bStoppingWeight3 := (iWeightCase = 20 AND P05_Weight.fbWeightStation.bWeighingCycleDone AND NOT P05_Weight.fbWeightStation.bCanReleaseForms);
bStoppingWeight4 := tonbCapSorterOrCapSorterDragError.Q; //Opóźnienie zeby wagi dkończyły cykl
//bStoppingWeight4 := stCapSorterRead.eError.bError OR P08_CapSorter.fbCapSorterDragStation.eState = E_Station.eError;

tonStoppingBottleTransfer1	(IN:=iBottleTransferCase = 2, PT:=T#3S);


IF stCapSorterRead.eError.bError THEN
	bCapSorterError := TRUE;
END_IF
tonbCapSorterError(IN:=bCapSorterError,	PT:=T#5S);


CASE iStoppingCase OF
	
	0: //init
		iStoppingCase										:= 10;
		
	10:
		IF
		//P01_BottleFeeder.fbBottleFeeder.eState<=10 AND					
		//P01_BottleFeeder.fbTurnTable.eState<=10 AND	
		//P01_BottleFeeder.fbGateBottleFeeder.eState<=13 AND
		//P01_PucksInserter.fbPucksInserter.eState<=10 AND					
		////P01_PucksInserter.fbTurnTable.eState<=10 AND	
		//P01_PucksInserter.fbGatePucksInserter.eState<=13 AND				
 		//(
		//stBottleSorterRead.ePackMLAutoState <> Tc3_PackML.E_PMLState.ePMLState_STOPPED OR
		//stBottleSorterRead.ePackMLAutoState <> Tc3_PackML.E_PMLState.ePMLState_IDLE OR
		//stBottleSorterRead.ePackMLAutoState <> Tc3_PackML.E_PMLState.ePMLState_RESETTING OR
		//stBottleSorterRead.ePackMLAutoState <> Tc3_PackML.E_PMLState.ePMLState_ABORTED OR
		//stBottleSorterRead.ePackMLAutoState <> Tc3_PackML.E_PMLState.ePMLState_ABORTING OR
		//NOT stBottleSorterRead.bEnable OR bBottleSorterDisable
		//) AND
		P01_Gates.fbGateBeforeDispencers.eState<=13 AND					
		P01_Gates.fbGateRobot.eState<=13 AND					
		P02_Dispencers.fbDispencersDragRightStation.eState<=10 AND
		P02_Dispencers.fbDispencersDragLeftStation.eState<=10 AND	
		P02_Dispencers.fbDispencer1.eState <= 10 AND
		P02_Dispencers.fbDispencer2.eState <= 10 AND
		P02_Dispencers.fbDispencer3.eState <= 10 AND
		P02_Dispencers.fbDispencer4.eState <= 10 AND
		P02_Dispencers.fbDispencersCatch1Station.eState <= 10 AND
		P02_Dispencers.fbDispencersCatch2Station.eState <= 10 AND
		P02_Dispencers.fbDispencersCatch3Station.eState <= 10 AND
		P02_Dispencers.fbDispencersCatch4Station.eState <= 10 AND	
		( //Namieszane na testy, kilka warunków
		bStoppingWeight1 OR
		// Nie ma Runa i nie ma nic na czujnikach
		bStoppingWeight2 OR	
		bStoppingWeight3 OR 
		//Bledy stacji
		bStoppingWeight4 OR
		//NOT bFormTransportersBeforeROPPCmdStart OR // Nowe do testów
		NOT bFormTransportersScrewerCmdStart OR
		(GeneralAlarms.nErrorCode = 61 AND  GeneralAlarms.bError)
		)	AND
		(	iWeightGateBeforeCASE = 50 OR iWeightGateBeforeCASE = 40 (*Szlaban wys.*) (*NOT Stoping*) OR 
			iWeightGateBeforeCASE = 20 (*Czeka na for. przed*) OR iWeightGateBeforeCASE = 30 OR NOT bWeightLiftEnable 
		) AND
		P05_Weight.fbWeight1.eState <= 10 AND
		P05_Weight.fbWeight2.eState <= 10 AND
		P05_Weight.fbWeight3.eState <= 10 AND
		P05_Weight.fbWeight4.eState <= 10 AND	
		P05_Weight.fbWeight5.eState <= 10 AND
		P05_Weight.fbWeight6.eState <= 10 AND			
		//P08_CapFeeder.fbCapFeeder.eState <= 10 AND		
		P06_LidFeeder.fbLidFeeder.eState <= 10 AND
		P06_LidFeeder.fbLidFeeder2.eState <= 10 AND
		P06_LidFeeder.fbLidFeederDragStation.eState <= 10 AND
		P06_LidPuttedCheck.fbLidPuttedCheck.eState <= 10 AND
		P06_LidSealer.fbLidSealer.eState <= 10 AND
		P06_LidSealer.fbLidSealer2.eState <= 10 AND
		P06_LidSealer.fbLidSealerDragStation.eState <= 10 AND
		
		(P06_WickFeeder.fbWickFeederSt.eRunningState1 = E_WickFeederState.eReady OR NOT VIS.bWickFeeder1Run) AND
		(P06_WickFeeder.fbWickFeederSt.eRunningState2 = E_WickFeederState.eReady OR NOT VIS.bWickFeeder2Run) AND	
		P06_WickFeeder.fbWickFeederDragStation.eState <= 10 AND
		
	
		//P07_ROPP.fbROPPFeeder.eState <= 10 AND
		//(P07_ROPP.fbROPPDrag.eState <= 10 OR (P07_ROPP.fbROPPDrag.eRunningState = E_DragStationState.eLifting AND NOT P07_ROPP.fbROPPDrag.bRun)) AND
		//P07_ROPP.fbROPPCapping.eState <= 10 AND
        //
		//(P08_CapSorter.fbCapSorterDragStation.eState <= 10 OR (P08_CapSorter.fbCapSorterDragStation.eRunningState = E_DragStationState.eLifting AND NOT P08_CapSorter.fbCapSorterDragStation.bRun)) AND 		
		//(
		//stCapSorterRead.ePackMLAutoState <> Tc3_PackML.E_PMLState.ePMLState_STOPPED OR
		//stCapSorterRead.ePackMLAutoState <> Tc3_PackML.E_PMLState.ePMLState_IDLE OR
		//stCapSorterRead.ePackMLAutoState <> Tc3_PackML.E_PMLState.ePMLState_RESETTING OR
		//stCapSorterRead.ePackMLAutoState <> Tc3_PackML.E_PMLState.ePMLState_ABORTED OR
		//stCapSorterRead.ePackMLAutoState <> Tc3_PackML.E_PMLState.ePMLState_ABORTING OR
		//NOT gvlCommunication.stCapSorterRead.bEnable OR bCapSorterDisable
		//) AND
		//(
		//	(iCapSorterCase <= 3 OR tonbCapSorterError.Q)
		//)	AND	
		P10_GripperScrewer.fb2GripperScrewer1.eState <= 10 AND
		P10_GripperScrewer.fb2GripperScrewer2.eState <= 10 AND		
		(P10_GripperScrewer.fbGripperScrewersDragStation.eState <= 10 OR (P10_GripperScrewer.fbGripperScrewersDragStation.eRunningState = E_DragStationState.eLifting AND NOT P10_GripperScrewer.fbGripperScrewersDragStation.bRun)) AND
		(P10_GripperScrewer.fbGripperScrewer1CatchStation.eState <= 10 OR P10_GripperScrewer.fb2GripperScrewer1.eState = 3 (*Error*) )	AND
		(P10_GripperScrewer.fbGripperScrewer2CatchStation.eState <= 10 OR P10_GripperScrewer.fb2GripperScrewer2.eState = 3 (*Error*) )	AND 
		P13_BottleTransfer.fbBottleTransfer.eState <= 10 AND
		(
		(iRobotPickCase = 10 OR iRobotPickCase = 20 OR iRobotPickCase = 220) OR  (*//Czeka na formatki*) 
		((iRobotPickCase = 210 OR iRobotPickCase = 210) AND  tonCycleBadBottleConveyorFullSensor2.Q ) OR  (*//Czeka nna wolne miejsce na odrzucie*) 		
		(iBottleTransferCase = 4 OR iBottleTransferCase = 1  OR tonStoppingBottleTransfer1.Q) (*Wypuscil formatki*)
		) // AND
		//P15_FormTransporters.fbFormTransporterScrewer.eState<=13 AND
		//P15_FormTransporters.fbFormTransporterDispencer.eState <= 13 AND
		//P15_FormTransporters.fbFormTransporterBeforeScrewer.eState <= 13
		THEN
			bFormTransportersScrewerCmdStart:=FALSE;
			VIS.bBottleFeederRun:=FALSE;
			bBottleFeederFormGateRun:=FALSE;
			VIS.bPucksInserterRun:=FALSE;
			//Vasyl 27.04 Stół podający
			bPucksInserterPushTable_m1_Run:=FALSE;
			bPucksInserterPushTable_m2_Run:=FALSE;
			bPucksInserterPushTable_m3_Run:=FALSE;
			//	
			bPucksInserterFormGateRun:=FALSE;			
			VIS.bGateBeforeDispencersRun:=FALSE;
			(*BottleSorter*)
			(*nic nie bedzie*)			
			VIS.bDispencer1Dose := FALSE;
			VIS.bDispencer2Dose := FALSE;
			VIS.bDispencer3Dose := FALSE;
			VIS.bDispencer4Dose := FALSE;
			VIS.bFormsDragingRightRun:=FALSE;
			GVL.bFormsDragingRightPrepareRun:=FALSE;
			VIS.bFormsDragingLeftRun:=FALSE;
			GVL.bFormsDragingLeftPrepareRun:=FALSE;
			VIS.bDispencers1Catch := FALSE;
			VIS.bDispencers2Catch := FALSE;
			VIS.bDispencers3Catch := FALSE;
			VIS.bDispencers4Catch := FALSE;
			VIS.bWeight1DoWeighting := FALSE;
			VIS.bWeight2DoWeighting := FALSE;
			VIS.bWeight3DoWeighting := FALSE;
			VIS.bWeight4DoWeighting := FALSE;
			VIS.bWeight5DoWeighting := FALSE;
			VIS.bWeight6DoWeighting := FALSE;
			VIS.bWeightLiftRun:=FALSE;
			bWeightLift2PhaseRun:=FALSE;
			bCapPuttedCheckRun	:=FALSE;
			VIS.bCapFeederRun := FALSE;
			VIS.bWickFeederSorterRun:=FALSE;
			VIS.bLidFeeder1Run := FALSE;	
			VIS.bLidFeeder2Run := FALSE;
			bLidFeederFormPositioningRun := FALSE;
			VIS.bLidFeederDragingStationRun := FALSE;	
			VIS.bLidPuttedCheckRun := FALSE;	
			VIS.bLidSealer1Run := FALSE;	
			VIS.bLidSealer2Run := FALSE;	
			VIS.bLidSealerDragingStationRun := FALSE;	

			VIS_ROPP.bROPPFeederRun		:=	FALSE;
			bROPPDragPrepareRun			:=	FALSE;
			VIS_ROPP.bROPPDragRun		:=	FALSE;
			bROPPCappingRunEngine		:=	FALSE;	
			VIS_ROPP.bROPPCappingRun1	:=	FALSE;					
			VIS_ROPP.bROPPCappingRun2	:=	FALSE;										
					
			bCapSorterRobotPlace:= FALSE;			
			bCapSorterRobotBottleAndNoCap1:= FALSE;
			bCapSorterRobotBottleAndNoCap2:= FALSE;	
			bCapSorterRobotBottleAndNoCap3:= FALSE;	
			bCapSorterRobotBottleAndNoCap4:= FALSE;	
			bCapSorterRobotPreparePlace	:= FALSE;			
			bCapSorterBeforeRobotBottleAndNoCap1	:=FALSE;	
			bCapSorterBeforeRobotBottleAndNoCap2	:=FALSE;	
			bCapSorterBeforeRobotBottleAndNoCap3	:=FALSE;	
			bCapSorterBeforeRobotBottleAndNoCap4	:=FALSE;	
			bGripperScrewer1Catch := FALSE;
			bGripperScrewer2Catch := FALSE;	
			VIS.bGripperScrewer1Run:=FALSE; 
			VIS.bGripperScrewer2Run:=FALSE;
			VIS.bGateRobotEntranceRun:=FALSE;
			VIS.bBottleDragingStationRun:=FALSE;
			GVL.bBottleDragingStationPrepareRun:=FALSE;
			VIS.bBottleTransferRun:=FALSE;
			
			iStoppingCase	:=	iStoppingCase	+	10;
	END_IF
			
	20:
	
		bFormTransportersDispencerCmdStart:=FALSE;	
		bFormTransportersAfterCapSorterCmdStart:=FALSE;
		bFormTransportersAfterScrewerCmdStart:=FALSE;	

		IF 	P14_BadBottleConyevor.fbBadBottleConveyor.eState <= 10 THEN
			bFormTransportersBeforeScrewerCmdStart:=FALSE;
			//bBadBottleConveyorStart:=FALSE;
			//bBadBottleConveyorStartTriggerDelay:=FALSE;
			iStoppingCase	:=	iStoppingCase	+	10;
			ACT_ResetCommands();
		END_IF

	30:
		ACT_ResetCommands();
		iStoppingCase											:= 0;
		fbPMLAuto.StateComplete									:= TRUE; 
		fbPMLManual.StateComplete								:= TRUE;	
			
END_CASE
END_ACTION

ACTION ACT_XtsChangeMode:

END_ACTION

ACTION aP00_SingleRealeseIfNoCapBeforeScrewers:
		
ulSingleRealeseIfNoCapFromScrewersNumber;
bSingleRealeseIfNoCapFromScrewersPulse;
iSingleRealeseIfNoCapFromScrewersPulse;

tonSingleRealeseIfNoCapFromScrewers1(IN:= iCaseSingleRealeseIfNoCapFromScrewersPulse = 20 AND (NOT P13_BottleTransfer.IbFirstFormCheckFormSensor OR NOT P13_BottleTransfer.IbSecondFormCheckFormSensor), PT:=T#3S);
tonSingleRealeseIfNoCapFromScrewers2 (IN:= P13_BottleTransfer.IbBottleTransferFormAfterSensor, PT:=T#3S);

rtSingleRealeseIfNoCapFromScrewers1 (CLK:= (eBeforeScrewers2PackageState[2].bBottlePresent AND NOT eBeforeScrewers2PackageState[2].bCapOK AND bCapPuttedCheckEnable) ,Q=>);
rtSingleRealeseIfNoCapFromScrewers2 (CLK:= (eBeforeScrewers2PackageState[1].bBottlePresent AND NOT eBeforeScrewers2PackageState[1].bCapOK AND bCapPuttedCheckEnable) ,Q=>);

IF rtSingleRealeseIfNoCapFromScrewers1.Q THEN
	iSingleRealeseIfNoCapFromScrewersPulse	:=	iSingleRealeseIfNoCapFromScrewersPulse	+	1;
	bSingleRealeseIfNoCapFromScrewersPulse	:=	TRUE;
ELSIF rtSingleRealeseIfNoCapFromScrewers2.Q THEN 
	iSingleRealeseIfNoCapFromScrewersPulse	:=	iSingleRealeseIfNoCapFromScrewersPulse	+	1;
	bSingleRealeseIfNoCapFromScrewersPulse	:=	TRUE;
END_IF

IF VIS.bSingleRealeseIfNoCapFromScrewers THEN

	CASE iCaseSingleRealeseIfNoCapFromScrewersPulse OF
		
		0:	//Brak nakretki
			IF bSingleRealeseIfNoCapFromScrewersPulse THEN
				iCaseSingleRealeseIfNoCapFromScrewersPulse	:=	iCaseSingleRealeseIfNoCapFromScrewersPulse	+	10;						
			END_IF
		
		10: //Blokuj przeciaganie 
			bSingleRealeseIfNoCapFromScrewersPulse			:= FALSE;
			bSingleRealeseIfNoCapFromScrewersDragBlock		:= TRUE;
			iCaseSingleRealeseIfNoCapFromScrewersPulse	:=	iCaseSingleRealeseIfNoCapFromScrewersPulse	+	10;

		20: //Czekaj na pustego robota
			IF tonSingleRealeseIfNoCapFromScrewers1.Q OR tonSingleRealeseIfNoCapFromScrewers2.Q THEN
				iCaseSingleRealeseIfNoCapFromScrewersPulse	:=	iCaseSingleRealeseIfNoCapFromScrewersPulse	+	10;
			END_IF			
			IF bSingleRealeseIfNoCapFromScrewersPulse THEN
				iCaseSingleRealeseIfNoCapFromScrewersPulse := 0;
			END_IF
			
		30: //Przeciągaj
			bSingleRealeseIfNoCapFromScrewersDragBlock		:=	FALSE;
			iCaseSingleRealeseIfNoCapFromScrewersPulse		:=	iCaseSingleRealeseIfNoCapFromScrewersPulse	+	10;
		
		40: //Czekaj na ten numer RFID i wyłaćz
			iCaseSingleRealeseIfNoCapFromScrewersPulse		:=	0;
		
	
	END_CASE
	
ELSE
	
	iCaseSingleRealeseIfNoCapFromScrewersPulse := 0;
END_IF
END_ACTION

ACTION aP01_Barriers:
//Załączenie szlabanów jak włączone jest dozowanie dwufazowe

IF bDosingTwoPhases THEN		
	GVL.bBarrierWeightRun:=TRUE;
	GVL.bBarrierDispencerRun:=TRUE;
ELSE	
	GVL.bBarrierWeightRun:=FALSE;
	GVL.bBarrierDispencerRun:=FALSE;
END_IF;
END_ACTION

ACTION aP01_BottleFeeder:
rttonDelayAfterStart(CLK:=tonDelayAfterStart.Q , Q=>);
IF rttonDelayAfterStart.Q THEN
	eBottleFeederPackageState[1].bBottlePresent	:=	TRUE;
END_IF
tontonDelayAfterStart(IN:=tonDelayAfterStart.Q , PT:=T#3S);

IF bBottleFeederEnable AND tonDelayAfterStart.Q  THEN

	bBottleFeederTurnTableRun							:=	TRUE;

	IF VIS.bWeighingForm OR VIS.bConfectionEnding OR NOT IbBottleFeederSafety THEN
		eBottleFeederPackageState[1].bBottlePresent	:=	TRUE;
	END_IF
	
	IF IbBottleFeederSafety AND NOT P01_BottleFeeder.fbBottleFeeder.bCycleDone  AND NOT eBottleFeederPackageState[1].bBottlePresent AND NOT (P00_PackML.fbPMLAuto.ePMLState = E_PMLState.ePMLState_STOPPING) 
	THEN
		VIS.bBottleFeederRun 							:=	tontonDelayAfterStart.Q;//TRUE; 
	END_IF
	
	IF (P01_BottleFeeder.fbBottleFeeder.bCycleDone OR eBottleFeederPackageState[1].bBottlePresent) AND NOT  P01_BottleFeeder.IbBottleFeederFormGateAfterSensor  THEN
		bBottleFeederFormGateRun						:=	TRUE;
	END_IF
	
	IF bBottleFeederFormGateRun AND P01_BottleFeeder.fbBottleFeeder.eRunningState >= E_BottleFeederState.eInsterting THEN
		eBottleFeederPackageState[1].bBottlePresent		:=	TRUE;
	END_IF
	
	IF P01_BottleFeeder.fbGateBottleFeeder.bCycleDone  THEN
		eBottleFeederPackageState[1].bBottlePresent		:=	FALSE;
		VIS.bBottleFeederRun 							:=	FALSE;
		bBottleFeederFormGateRun						:=	FALSE;
	END_IF

	IF (P00_PackML.fbPMLAuto.ePMLState = E_PMLState.ePMLState_STOPPING) THEN
		VIS.bBottleFeederRun 							:=	FALSE;
		bBottleFeederTurnTableRun						:=	FALSE;
	END_IF
	
END_IF
END_ACTION

ACTION aP01_BottleSorter:

END_ACTION

ACTION aP01_Gates:
iBeforeDispencerCounter			:=	BOOL_TO_INT(eBeforeDispencersPackageState[1].bFormPresent) +
						 			BOOL_TO_INT(eBeforeDispencersPackageState[2].bFormPresent) +
 						 			BOOL_TO_INT(eBeforeDispencersPackageState[3].bFormPresent) +
 						 			BOOL_TO_INT(eBeforeDispencersPackageState[4].bFormPresent);
						 
iBeforeDispencer2PhaseCounter	:= 	BOOL_TO_INT(eBeforeDispencer34PackageState2Phase[1].bFormPresent) +				 
						  			BOOL_TO_INT(eBeforeDispencer34PackageState2Phase[2].bFormPresent);

// Szlaban przed dozownikiem
CASE iGateDispCase OF
	
		0:
			//Kasowanie rozkazów
			VIS.bGateBeforeDispencersRun	:=	FALSE;
			iGateDispCase					:=	iGateDispCase	+	10;
			
		10: 
			//Opóźnienie startu
			IF tonDelayAfterStart.Q  AND NOT bPhaseChanging THEN
				iGateDispCase				:=	iGateDispCase	+	10;
			END_IF
	
		20:
			// Kontrola po uruchomineiu
			// Zajęty czujnik przed i za  bramką //Zamknij
			IF MAIN.IbFourthFormCheckFormSensor AND MAIN.IbFormCheckFormSensor THEN
				iGateDispCase:=100;
			END_IF
			
			//Zajęty czujnika przed bramką, ale pusty przy 4 formatce //Wpuszczanie pojedynczo
			IF NOT MAIN.IbFourthFormCheckFormSensor AND MAIN.IbFormCheckFormSensor THEN
				iGateDispCase:=200;
			END_IF
			
			//brak formatek przy obydwu czujnikach //Wpuszczanie razem
			IF NOT MAIN.IbFourthFormCheckFormSensor AND NOT MAIN.IbFormCheckFormSensor THEN
				iGateDispCase:=200;
			END_IF	
	
		100: //Zamkniecie szlbanu
			VIS.bGateBeforeDispencersRun:=FALSE;
			iGateDispCase:=400;
			
		200: //Wpuszczanie pojedynczo		
			tonWeightBeforeGateDispSensor();
			tonWeightBeforeGateDispSensor.IN:=NOT MAIN.IbFourthFormCheckFormSensor AND MAIN.IbFormCheckFormSensor AND NOT VIS.bGateBeforeDispencersRun;
			tonWeightBeforeGateDispSensor.PT:=T#1S;
			
			
			//Otwarcie szlabanu
			IF tonWeightBeforeGateDispSensor.Q AND (bPhaseChangingGatePermission OR NOT brtLongDelayFirstDragingDone OR bLongDelayAfterStart) AND NOT tonQueAfterPlatin.Q THEN
				VIS.bGateBeforeDispencersRun	:=	TRUE;
			END_IF
			// Otwarcie szlabanu jak nie ma formatek przez dłuższy czas przy rozpoczęciu konfekcji dodane 06.06
		
			IF tonCheckFormBeforeDispencersGate.Q AND NOT VIS.bGateBeforeDispencersRun THEN
				VIS.bGateBeforeDispencersRun	:=	TRUE;
			END_IF
			
			//Zamknieceie szlabanu
			IF P01_Gates.fbGateBeforeDispencers.bCycleDone THEN // ZMIANA NA CYCLE DONE - MUSI DZIALAĆ
				VIS.bGateBeforeDispencersRun	:=	FALSE;
			END_IF

			
			tonBeforeGateSensorDelay();
			tonBeforeGateSensorDelay.IN:= MAIN.IbFourthFormCheckFormSensor(* AND MAIN.IbFormCheckFormSensor*);
			tonBeforeGateSensorDelay.PT:=T#5S;
			
			IF tonBeforeGateSensorDelay.Q  THEN
				tonBeforeGateSensorDelay();
				tonBeforeGateSensorDelay.IN:=FALSE;
				iGateDispCase:=320;
			END_IF
			
		300:
			VIS.bGateBeforeDispencersRun:=TRUE;
			iGateDispCase:=400;
			
		320:	
			//Kasowanie rozkazów 
			VIS.bGateBeforeDispencersRun:=FALSE;
			IF iPhaseChangingStep<> 6 THEN
			iGateDispCase:=400;	
			END_IF
		400:
			IF ((iBeforeDispencerCounter=4 AND NOT bDosingTwoPhases) OR (iBeforeDispencer2PhaseCounter=2 AND bDosingTwoPhases)) AND tonLongDelayAfterStart.Q AND MAIN.IbFourthFormCheckFormSensor THEN
				 iGateDispCase:=500;
			END_IF
			
			IF ((iBeforeDispencerCounter<4 AND NOT bDosingTwoPhases)OR ( iBeforeDispencer2PhaseCounter<2 AND bDosingTwoPhases)) AND tonLongDelayAfterStart.Q (*AND MAIN.IbFormCheckFormSensor*) AND tonCheckFourthFormNotPresent.Q (*NOT MAIN.IbFourthFormCheckFormSensor *)(*AND P02_Dispencers.IbFormsDragHomePositionSensor *)THEN
				 iGateDispCase:=600;
			END_IF
			
		500:
			IF P01_Gates.fbGateBeforeDispencers.bCycleDone OR NOT VIS.bGateBeforeDispencersRun THEN 
				VIS.bGateBeforeDispencersRun	:=	FALSE;
				iGateDispCase					:=	800;
			END_IF
			
		600:
			IF NOT 	P01_Gates.fbGateBeforeDispencers.bCycleDone THEN
				VIS.bGateBeforeDispencersRun:=TRUE;
			END_IF
			
			IF ((iBeforeDispencerCounter=4 AND NOT bDosingTwoPhases) OR (iBeforeDispencer2PhaseCounter=2 AND bDosingTwoPhases)) THEN 
				VIS.bGateBeforeDispencersRun	:=	FALSE;
				iGateDispCase					:=	800;
			END_IF
			
			IF P00_PackML.fbPMLAuto.ePMLState = E_PMLState.ePMLState_STOPPING THEN
				iGateDispCase:=800;
			END_IF	
			
			
		800:
			 IF NOT (P00_PackML.fbPMLAuto.ePMLState = E_PMLState.ePMLState_STOPPING) THEN
				iGateDispCase:=320;
			END_IF
				
			IF P00_PackML.fbPMLAuto.ePMLState = E_PMLState.ePMLState_STOPPING THEN
				VIS.bGateBeforeDispencersRun:=FALSE;
			END_IF	
END_CASE
END_ACTION

ACTION aP01_GatesLidFeederBarrier:


VIS.bBarrierLidFeederRun;

IF tonLongDelayAfterStart.Q AND (bLidFeederEnable OR bWickFeederEnable) THEN
	IF tonDelayAfterStart.Q THEN
		VIS.bBarrierLidFeederRun	:= TRUE;
	END_IF
ELSIF NOT bLidFeederEnable AND NOT bWickFeederEnable THEN
	VIS.bBarrierLidFeederRun		:= FALSE;
END_IF

//Dodane po zatrzymaniu awaryjnym bramka się podnosi. Jak jest czujnik i załączona to zostaje opuszczona
IF (bLidFeederEnable OR bWickFeederEnable) AND P01_Gates.IbLidFeederBarrierOnSensor THEN
	VIS.bBarrierLidFeederRun	:= TRUE;
END_IF
END_ACTION

ACTION aP01_PucksInserter:
rttonDelayAfterStart(CLK:=tonDelayAfterStart.Q , Q=>);
IF rttonDelayAfterStart.Q THEN
	//IF NOT P01_PucksInserter.QbPucksInserterFormGate THEN
	//	bPucksInserterFormGateRun := TRUE;
	//END_IF
	eBottleFeederPackageState[1].bBottlePresent	:=	TRUE;
END_IF
tontonDelayAfterStart(IN:=tonDelayAfterStart.Q , PT:=T#3S);
tonDelayForGatePI(IN:=P01_PucksInserter.IbPucksInserterFormGateAfterSensor, PT:=T#500MS);
fbIbPucksInserterFormGateAfterSensor(bIN:=P01_PucksInserter.IbPucksInserterFormGateAfterSensor, tFilterTimeon:=T#300MS, tFilterTimeOff:=T#100MS);
//tonPucksInserterPushTableOff(IN:= "CZUJNIK KOLEJKI NA STOLE", PT:=(UDINT_TO_TIME(VIS.udiPucksInserterPushTableOFFDelayShow)));

IF bFormTransportersDispencerSlowSpeed THEN
	iPucksInserterFormGateDelayAdd := 400;
ELSE
	iPucksInserterFormGateDelayAdd := 0;
END_IF


IF bPucksInserterEnable AND tonDelayAfterStart.Q  THEN

	bPucksInserterTurnTableRun							:=	TRUE;

	//IF VIS.bWeighingForm OR VIS.bConfectionEnding THEN // Przeniesione do PI
	//	eBottleFeederPackageState[1].bBottlePresent	:=	TRUE;
	//END_IF
	
	IF  NOT P01_PucksInserter.fbPucksInserter.bCycleDone  AND NOT eBottleFeederPackageState[1].bBottlePresent AND NOT (P00_PackML.fbPMLAuto.ePMLState = E_PMLState.ePMLState_STOPPING) 
	THEN
		VIS.bPucksInserterRun 							:=	tontonDelayAfterStart.Q;//TRUE; 
	END_IF
	
	IF (P01_PucksInserter.fbPucksInserter.bCycleDone OR eBottleFeederPackageState[1].bBottlePresent) AND NOT fbIbPucksInserterFormGateAfterSensor.bOut THEN //NOT  P01_PucksInserter.IbPucksInserterFormGateAfterSensor  THEN
		bPucksInserterFormGateRun						:=	TRUE;
	END_IF
	IF P01_PucksInserter.fbPucksInserter.eRunningState = E_PuckInserterState.eInsterting THEN
		eBottleFeederPackageState[1].bBottlePresent		:=	FALSE;
	END_IF	
	IF bPucksInserterFormGateRun AND P01_PucksInserter.fbPucksInserter.eRunningState >= E_PuckInserterState.eBackToPosition THEN
		eBottleFeederPackageState[1].bBottlePresent		:=	TRUE;
	END_IF
	
	IF P01_PucksInserter.fbGatePucksInserter.bCycleDone  AND NOT P01_PucksInserter.IbPucksInserterFormGateBeforeSensor THEN
		eBottleFeederPackageState[1].bBottlePresent		:=	FALSE;
		VIS.bPucksInserterRun 							:=	FALSE;
		bPucksInserterFormGateRun						:=	FALSE;
	END_IF

	IF (P00_PackML.fbPMLAuto.ePMLState = E_PMLState.ePMLState_STOPPING) THEN
		VIS.bPucksInserterRun 							:=	FALSE;
		bPucksInserterTurnTableRun						:=	FALSE;
		bPucksInserterPushTable_m1_Run					:=	FALSE;
		bPucksInserterPushTable_m2_Run					:=	FALSE;
		bPucksInserterPushTable_m3_Run					:=	FALSE;
	END_IF
ELSE
	// SAM SZLABAN
	tonIbPucksInserterFormGateBeforeSensor (IN:=P01_PucksInserter.IbPucksInserterFormGateBeforeSensor , PT:=T#300MS);
	IF tonDelayAfterStart.Q  THEN
		P01_PucksInserter.IbPucksInserterFormGateBeforeSensor;
		GVL.bFormTransportersDispencerCmdStart;
		P01_PucksInserter.fbGatePucksInserter.bCycleDone;
		
		IF P01_PucksInserter.IbPucksInserterFormGateBeforeSensor AND NOT P01_PucksInserter.fbGatePucksInserter.bCycleDone AND NOT fbIbPucksInserterFormGateAfterSensor.bOut THEN 
			bPucksInserterFormGateRun						:=	TRUE;
		END_IF
	
		IF bPucksInserterFormGateRun AND P01_PucksInserter.fbGatePucksInserter.bCycleDone THEN
			bPucksInserterFormGateRun						:=	FALSE;
		END_IF
	END_IF
END_IF
(*
udiPucksInserterPushTable_m1_VelocitySV:=VIS.udiPucksInserterPushTableVelocityShow;		
iPucksInserterPushTable_m2_VelocitySV:=VIS.iPucksInserterPushTableRollersVelocityShow;	
udiPucksInserterPushTableActuatorPUSHDelay:=VIS.udiPucksInserterPushTableActuatorPUSHDelayShow;
udiPucksInserterPushTableActuatorPULLDelay:=VIS.udiPucksInserterPushTableActuatorPULLDelayShow;
udiPucksInserterPushTableOFFDelay	:= VIS.udiPucksInserterPushTableOFFDelayShow;
bPucksInserterPushTableGateRun		 :=VIS.bPucksInserterPushTableActuatorEnableShow;	
bPucksInserterPushTable_m2_Enable	 :=VIS.bPucksInserterPushTableRollerEnableShow;		
bPucksInserterPushTable_m1_Enable	 :=VIS.bPucksInserterPushTableEnableShow;
*)
fbIbPucksInserterPushTablesSensor(bIN:=NOT P01_PucksInserter.IbPucksInserterPushTablesSensor AND P01_PucksInserter.uiPucksInserterConveyorActualVelocity>100, tFilterTimeon:=T#3S, tFilterTimeOff:=T#6S);

IF bPucksInserterEnable AND tonDelayAfterStart.Q THEN

	bPucksInserterPushTable_m1_Run := fbIbPucksInserterPushTablesSensor.bOut;
	bPucksInserterPushTable_m2_Run := fbIbPucksInserterPushTablesSensor.bOut;
	bPucksInserterPushTable_m3_Run := fbIbPucksInserterPushTablesSensor.bOut;

END_IF
END_ACTION

ACTION aP02_BottlePusher:
P02_BottlePusher.IbBottlePusherBottleBeforeSensor;


(*1*)
IF P02_BottlePusher.IbBottlePusherBottleBeforeSensor THEN 
	bBottlePusherBottleBeforeSensor := TRUE;
END_IF

(*2*)
tonBottlePusherBottleBeforeSensor	(IN:=bBottlePusherBottleBeforeSensor,	PT:=T#0MS);
IF tonBottlePusherBottleBeforeSensor.Q THEN
	VIS.bBottlePusherRun	:= TRUE;
END_IF

(*3*)
IF P02_BottlePusher.fbBottlePusher.bCycleDone THEN
	VIS.bBottlePusherRun			:= FALSE;
	bBottlePusherBottleBeforeSensor	:=	FALSE;
END_IF
END_ACTION

ACTION aP02_Dispencers1Phase:
// - Aborted wyżej

(***********************************)
(**********P02_Dispencers***********)


tonDosingDelay				(IN:=iDispencersCase=4
								,PT:=UINT_TO_TIME(uiDispencerStartDosingDelay+300));//Opoznienie przed dozowaniem //Check
tonCatchDelay				(IN:=iDispencersCase=4
								,PT:=UINT_TO_TIME(uiDispencerStartDosingDelay));//Opoznienie przed dozowaniem //Check
								
								
tonErrorDosing1					(IN:=VIS.bDispencer1Dose, PT:=T#20S);//Timer za długiego dozowania
tonErrorDosing2					(IN:=VIS.bDispencer2Dose, PT:=T#20S);
tonErrorDosing3					(IN:=VIS.bDispencer3Dose, PT:=T#20S);
tonErrorDosing4					(IN:=VIS.bDispencer4Dose, PT:=T#20S);

bDisp1FormsAndNoBottle			 := eDispencersPackageState[1].bFormPresent AND NOT eDispencersPackageState[1].bBottlePresent ;//Sygnały chytaków bez butelek
bDisp2FormsAndNoBottle			 := eDispencersPackageState[2].bFormPresent AND NOT eDispencersPackageState[2].bBottlePresent;
bDisp3FormsAndNoBottle			 := eDispencersPackageState[3].bFormPresent AND NOT eDispencersPackageState[3].bBottlePresent;
bDisp4FormsAndNoBottle			 := eDispencersPackageState[4].bFormPresent AND NOT eDispencersPackageState[4].bBottlePresent;

	tonDispencersCase4Delay(IN:=iDispencersCase=4,PT:=T#100MS);

//Sygnał zakończenia dozowania
tonbDosingDone (IN:= bDosingDone OR bDosingDoneFaster, PT:=T#20MS);
bDosingDone  := 				(	NOT bDispencer1Enable OR eDispencersPackageState[1].bDoseAborted OR	
																(
																(VIS.bDispencer1Dose AND (P02_Dispencers.fbDispencer1.bCycleDone OR tonErrorDosing1.Q))  OR 
																NOT VIS.bDispencer1Dose
																)  
								)  AND 
								(	NOT bDispencer2Enable OR eDispencersPackageState[2].bDoseAborted OR 
																(
																(VIS.bDispencer2Dose AND (P02_Dispencers.fbDispencer2.bCycleDone  OR tonErrorDosing2.Q)) OR
																 NOT VIS.bDispencer2Dose
																)  
								)  AND 
								(	NOT bDispencer3Enable OR eDispencersPackageState[3].bDoseAborted OR 
																(
																(VIS.bDispencer3Dose AND (P02_Dispencers.fbDispencer3.bCycleDone  OR tonErrorDosing3.Q)) OR
																 NOT VIS.bDispencer3Dose
																)  
								)  AND 
								(	NOT bDispencer4Enable OR eDispencersPackageState[4].bDoseAborted OR 
																(
																(VIS.bDispencer4Dose AND (P02_Dispencers.fbDispencer4.bCycleDone  OR tonErrorDosing4.Q)) OR
																 NOT VIS.bDispencer4Dose
																)  
								)  AND 
								( iDispencersCase = 4 AND tonDosingDelay.Q) AND 
								(
									tonCatchNotEnable.Q OR tonCatched.Q OR 
									(bDisp1FormsAndNoBottle AND bDisp2FormsAndNoBottle AND bDisp3FormsAndNoBottle AND bDisp4FormsAndNoBottle) OR 
									(NOT bDispencer1Enable AND NOT bDispencer2Enable AND NOT bDispencer3Enable AND NOT bDispencer4Enable) 
								);
								
bDosingDoneFaster:=		    (tonCatched.Q AND 																											//Dorobilem bottle present
								 ((VIS.bDispencer1Dose AND P02_Dispencers.QbDispencer1DropCatcherValveActuator) OR NOT bDispencer1Enable OR NOT eDispencersPackageState[1].bBottlePresent)
                                  AND
                                  ((VIS.bDispencer2Dose AND P02_Dispencers.QbDispencer2DropCatcherValveActuator) OR NOT bDispencer2Enable OR NOT eDispencersPackageState[2].bBottlePresent)                                                                                               (*Dodano szybsze otwieranie szlabanu jak tylko tacki się zamkną*)                     
                                  AND
                                  ((VIS.bDispencer3Dose AND P02_Dispencers.QbDispencer3DropCatcherValveActuator) OR NOT bDispencer3Enable OR NOT eDispencersPackageState[3].bBottlePresent)
                                  AND
                                  ((VIS.bDispencer4Dose AND P02_Dispencers.QbDispencer4DropCatcherValveActuator) OR NOT bDispencer4Enable OR NOT eDispencersPackageState[4].bBottlePresent)                                                                                               (*Dodano szybsze otwieranie szlabanu jak tylko tacki się zamkną*)                     
                                 		  
								  
								  
                			 ) (************************ tutaj od podwojnej dozy******)
                   OR               // Dodanie jeżeli tacki się nie wysuwają to przesuwaj szybciej jeżeli dozowniki są w zasysaniu
                   (               ((VIS.bDispencer1Dose AND	(P02_Dispencers.fbDispencer1.eRunningState = E_DispencerState.eSucking AND NOT P02_Dispencers.fbDispencer1.bDoSecondDose)) OR NOT bDispencer1Enable)
									 AND
									 ((VIS.bDispencer2Dose AND	(P02_Dispencers.fbDispencer2.eRunningState = E_DispencerState.eSucking AND NOT P02_Dispencers.fbDispencer2.bDoSecondDose)) OR NOT bDispencer2Enable)   
									 AND
									 ((VIS.bDispencer3Dose AND	(P02_Dispencers.fbDispencer3.eRunningState = E_DispencerState.eSucking AND NOT P02_Dispencers.fbDispencer3.bDoSecondDose)) OR NOT bDispencer3Enable)
									 AND
									 ((VIS.bDispencer4Dose AND	(P02_Dispencers.fbDispencer4.eRunningState = E_DispencerState.eSucking AND NOT P02_Dispencers.fbDispencer4.bDoSecondDose)) OR NOT bDispencer4Enable)
                   );						
													
bDispencersReady := 			(NOT bDispencer1Enable OR P02_Dispencers.fbDispencer1.eState = E_Station.eReady) AND 
								(NOT bDispencer2Enable OR P02_Dispencers.fbDispencer2.eState = E_Station.eReady) AND	
								(NOT bDispencer3Enable OR P02_Dispencers.fbDispencer3.eState = E_Station.eReady) AND
								(NOT bDispencer4Enable OR P02_Dispencers.fbDispencer4.eState = E_Station.eReady) AND																	
								(
								NOT bDispencersCatchEnable OR (NOT bDispencer1Enable AND NOT bDispencer2Enable AND NOT bDispencer3Enable AND NOT bDispencer4Enable) OR 
								(
									(P02_Dispencers.fbDispencersCatch1Station.eState=E_Station.eReady AND NOT P02_Dispencers.fbDispencersCatch1Station.bCycleDone) AND
									(P02_Dispencers.fbDispencersCatch2Station.eState=E_Station.eReady AND NOT P02_Dispencers.fbDispencersCatch2Station.bCycleDone) AND
									(P02_Dispencers.fbDispencersCatch3Station.eState=E_Station.eReady AND NOT P02_Dispencers.fbDispencersCatch3Station.bCycleDone) AND
									(P02_Dispencers.fbDispencersCatch4Station.eState=E_Station.eReady AND NOT P02_Dispencers.fbDispencersCatch4Station.bCycleDone) 
								)
								);											
					(************************ tutaj od podwojnej dozy******)
bDispencersReadyOrSucking := 	(NOT bDispencer1Enable OR P02_Dispencers.fbDispencer1.eState = E_Station.eReady OR (P02_Dispencers.fbDispencer1.eRunningState = E_DispencerState.eSucking AND NOT P02_Dispencers.fbDispencer1.bDoSecondDose) OR (P02_Dispencers.fbDispencer1.eRunningState = E_DispencerState.eGoingUp	AND P02_Dispencers.QbDispencer1DropCatcherValveActuator)) AND 
								(NOT bDispencer2Enable OR P02_Dispencers.fbDispencer2.eState = E_Station.eReady OR (P02_Dispencers.fbDispencer2.eRunningState = E_DispencerState.eSucking AND NOT P02_Dispencers.fbDispencer2.bDoSecondDose) OR (P02_Dispencers.fbDispencer2.eRunningState = E_DispencerState.eGoingUp	AND P02_Dispencers.QbDispencer2DropCatcherValveActuator)) AND
								(NOT bDispencer3Enable OR P02_Dispencers.fbDispencer3.eState = E_Station.eReady OR (P02_Dispencers.fbDispencer3.eRunningState = E_DispencerState.eSucking AND NOT P02_Dispencers.fbDispencer3.bDoSecondDose) OR (P02_Dispencers.fbDispencer3.eRunningState = E_DispencerState.eGoingUp	AND P02_Dispencers.QbDispencer3DropCatcherValveActuator)) AND
								(NOT bDispencer4Enable OR P02_Dispencers.fbDispencer4.eState = E_Station.eReady OR (P02_Dispencers.fbDispencer4.eRunningState = E_DispencerState.eSucking AND NOT P02_Dispencers.fbDispencer4.bDoSecondDose) OR (P02_Dispencers.fbDispencer4.eRunningState = E_DispencerState.eGoingUp	AND P02_Dispencers.QbDispencer4DropCatcherValveActuator));
bCatchersReady:=		NOT bDispencersCatchEnable OR (NOT bDispencer1Enable AND NOT bDispencer2Enable AND NOT bDispencer3Enable AND NOT bDispencer4Enable) OR 
								(
									(P02_Dispencers.fbDispencersCatch1Station.eState=E_Station.eReady AND NOT P02_Dispencers.fbDispencersCatch1Station.bCycleDone) AND
									(P02_Dispencers.fbDispencersCatch2Station.eState=E_Station.eReady AND NOT P02_Dispencers.fbDispencersCatch2Station.bCycleDone) AND
									(P02_Dispencers.fbDispencersCatch3Station.eState=E_Station.eReady AND NOT P02_Dispencers.fbDispencersCatch3Station.bCycleDone) AND
									(P02_Dispencers.fbDispencersCatch4Station.eState=E_Station.eReady AND NOT P02_Dispencers.fbDispencersCatch4Station.bCycleDone) 
								)			;
																
//Timer braku chwytania opakowania (************************ tutaj od podwojnej dozy******)
tonCatchNotEnable				(IN:=NOT bDispencersCatchEnable AND 
								(
									VIS.bDispencer1Dose OR VIS.bDispencer2Dose OR VIS.bDispencer3Dose OR VIS.bDispencer4Dose OR 
									(
									((P02_Dispencers.fbDispencer1.eRunningState = E_DispencerState.eSucking AND NOT P02_Dispencers.fbDispencer1.bDoSecondDose) OR NOT bDispencer1Enable) OR 
									((P02_Dispencers.fbDispencer2.eRunningState = E_DispencerState.eSucking AND NOT P02_Dispencers.fbDispencer2.bDoSecondDose) OR NOT bDispencer2Enable) OR
									((P02_Dispencers.fbDispencer3.eRunningState = E_DispencerState.eSucking AND NOT P02_Dispencers.fbDispencer3.bDoSecondDose) OR NOT bDispencer3Enable) OR 
									((P02_Dispencers.fbDispencer4.eRunningState = E_DispencerState.eSucking AND NOT P02_Dispencers.fbDispencer4.bDoSecondDose) OR NOT bDispencer4Enable) 
									)
								),PT:=T#20MS);
//Opoznienie chwycenia
tonCatched						(IN:=	(P02_Dispencers.fbDispencersCatch1Station.eRunningState=E_CatchStationState.eCatched OR P02_Dispencers.fbDispencersCatch1Station.eRunningState=E_CatchStationState.eNotCatched OR  NOT eDispencersPackageState[1].bBottlePresent OR NOT bDispencer1Enable) AND
										(P02_Dispencers.fbDispencersCatch2Station.eRunningState=E_CatchStationState.eCatched OR P02_Dispencers.fbDispencersCatch2Station.eRunningState=E_CatchStationState.eNotCatched OR  NOT eDispencersPackageState[2].bBottlePresent OR NOT bDispencer2Enable) AND
										(P02_Dispencers.fbDispencersCatch3Station.eRunningState=E_CatchStationState.eCatched OR P02_Dispencers.fbDispencersCatch3Station.eRunningState=E_CatchStationState.eNotCatched OR  NOT eDispencersPackageState[3].bBottlePresent OR NOT bDispencer3Enable) AND
										(P02_Dispencers.fbDispencersCatch4Station.eRunningState=E_CatchStationState.eCatched OR P02_Dispencers.fbDispencersCatch4Station.eRunningState=E_CatchStationState.eNotCatched OR  NOT eDispencersPackageState[4].bBottlePresent OR NOT bDispencer4Enable)
										,PT:=T#500MS);
										
//Filtry sygnałów wykrywania butelek pod chwytakiem
bDispencer1CatchedOrNoBottle := P02_Dispencers.fbDispencersCatch1Station.eRunningState=E_CatchStationState.eCatched OR NOT eDispencersPackageState[1].bBottlePresent;
bDispencer2CatchedOrNoBottle := P02_Dispencers.fbDispencersCatch2Station.eRunningState=E_CatchStationState.eCatched OR NOT eDispencersPackageState[2].bBottlePresent;
bDispencer3CatchedOrNoBottle := P02_Dispencers.fbDispencersCatch3Station.eRunningState=E_CatchStationState.eCatched OR NOT eDispencersPackageState[3].bBottlePresent;
bDispencer4CatchedOrNoBottle := P02_Dispencers.fbDispencersCatch4Station.eRunningState=E_CatchStationState.eCatched OR NOT eDispencersPackageState[4].bBottlePresent;

fbDispencer1BottleInCatcherSensor(bIN:=P02_Dispencers.fbDispencersCatch1Station.eRunningState=E_CatchStationState.eCatched AND bDispencer2CatchedOrNoBottle AND IbEmergencyStop, tFilterTimeOn:=T#50MS, tFilterTimeOff:=T#100MS, bOUT=> );(*Filtr wejścia cyfrowego*)
fbDispencer2BottleInCatcherSensor(bIN:=P02_Dispencers.fbDispencersCatch2Station.eRunningState=E_CatchStationState.eCatched AND bDispencer1CatchedOrNoBottle AND IbEmergencyStop, tFilterTimeOn:=T#50MS, tFilterTimeOff:=T#100MS, bOUT=> );(*Filtr wejścia cyfrowego*)//bylo 150
fbDispencer3BottleInCatcherSensor(bIN:=P02_Dispencers.fbDispencersCatch3Station.eRunningState=E_CatchStationState.eCatched AND bDispencer4CatchedOrNoBottle AND IbEmergencyStop, tFilterTimeOn:=T#50MS, tFilterTimeOff:=T#100MS, bOUT=> );(*Filtr wejścia cyfrowego*)
fbDispencer4BottleInCatcherSensor(bIN:=P02_Dispencers.fbDispencersCatch4Station.eRunningState=E_CatchStationState.eCatched AND bDispencer3CatchedOrNoBottle AND IbEmergencyStop, tFilterTimeOn:=T#50MS, tFilterTimeOff:=T#500MS, bOUT=> );(*Filtr wejścia cyfrowego*)

CASE iDispencersCase OF

		0: //Kilka stanów niepotrzebnych, zeby zgadzało się z innymi liniami, w razie poprawek, aktualizacji
			iDispencersCase := 4;
			
		1:	//Przepisywanie danych po wydozowaniu
			
			VIS.bDispencers1Catch 	:=	FALSE;
			VIS.bDispencers2Catch 	:=	FALSE;
			VIS.bDispencers3Catch 	:=	FALSE;
			VIS.bDispencers4Catch 	:=	FALSE;	
			
			(**PRZEPISYWANIE PARAMETRÓW PO WYDOZOWANIU**)
			eDispencersPackageState[1].lrDoseVolumeCV					:= ABS(lrDosedMass1CVAux);
			eDispencersPackageState[1].lrDoseVolumeSV 					:= lrDispencer1DoseVolume + VIS.lrDispencer1CorrectionWeight;
			eDispencersPackageState[1].nDispencerNr 					:= 1;
			eDispencersPackageState[1].tDispencingTime 					:= P02_Dispencers.fbDispencer1.tCycleTime;
			eDispencersPackageState[2].lrDoseVolumeCV					:= ABS(lrDosedMass2CVAux);
			eDispencersPackageState[2].lrDoseVolumeSV 					:= lrDispencer1DoseVolume + VIS.lrDispencer2CorrectionWeight;
			eDispencersPackageState[2].nDispencerNr 					:= 2;
			eDispencersPackageState[2].tDispencingTime 					:= P02_Dispencers.fbDispencer2.tCycleTime;
	
			eDispencersPackageState[3].lrDoseVolumeCV					:= ABS(lrDosedMass3CVAux);
			eDispencersPackageState[3].lrDoseVolumeSV 					:= lrDispencer1DoseVolume + VIS.lrDispencer3CorrectionWeight;
			eDispencersPackageState[3].nDispencerNr 					:= 3;
			eDispencersPackageState[3].tDispencingTime 					:= P02_Dispencers.fbDispencer3.tCycleTime;
			eDispencersPackageState[4].lrDoseVolumeCV					:= ABS(lrDosedMass4CVAux);
			eDispencersPackageState[4].lrDoseVolumeSV 					:= lrDispencer1DoseVolume + VIS.lrDispencer4CorrectionWeight;
			eDispencersPackageState[4].nDispencerNr 					:= 4;
			eDispencersPackageState[4].tDispencingTime 					:= P02_Dispencers.fbDispencer4.tCycleTime;

			(*Sprawdzanie czy wydozowana ilość zgadza się z zadaną*)			
			IF 	ABS(eDispencersPackageState[1].lrDoseVolumeSV  - eDispencersPackageState[1].lrDoseVolumeCV) < 2 THEN 
					eDispencersPackageState[1].bDosed := TRUE;	ELSE
					eDispencersPackageState[1].bDoseAborted := TRUE;	
			END_IF
			IF 	ABS(eDispencersPackageState[2].lrDoseVolumeSV  - eDispencersPackageState[2].lrDoseVolumeCV) < 2 THEN 
					eDispencersPackageState[2].bDosed := TRUE;	ELSE
					eDispencersPackageState[2].bDoseAborted := TRUE;	
			END_IF
			IF 	ABS(eDispencersPackageState[3].lrDoseVolumeSV  - eDispencersPackageState[3].lrDoseVolumeCV) < 2 THEN 
					eDispencersPackageState[3].bDosed := TRUE;	ELSE
					eDispencersPackageState[3].bDoseAborted := TRUE;	
			END_IF
			IF 	ABS(eDispencersPackageState[4].lrDoseVolumeSV  - eDispencersPackageState[4].lrDoseVolumeCV) < 2 THEN 
					eDispencersPackageState[4].bDosed := TRUE;	ELSE
					eDispencersPackageState[4].bDoseAborted := TRUE;	
			END_IF
			(*******************)	
			
			IF NOT bDispencer1Enable THEN (*Jezeli dozowniki wylaczone to wpisz jakas wartość zeby platynki zakładało*)
				eDispencersPackageState[1].lrDoseVolumeCV 			:=3;
				eDispencersPackageState[1].bDosed					:= TRUE;				
				eDispencersPackageState[1].bDoseAborted				:= TRUE;
			END_IF
			IF NOT bDispencer2Enable THEN (*Jezeli dozowniki wylaczone to wpisz jakas wartość zeby platynki zakładało*)	
				eDispencersPackageState[2].lrDoseVolumeCV 			:=3;
				eDispencersPackageState[2].bDosed					:= TRUE;				
				eDispencersPackageState[2].bDoseAborted				:= TRUE;
			END_IF
			IF NOT bDispencer3Enable THEN (*Jezeli dozowniki wylaczone to wpisz jakas wartość zeby platynki zakładało*)
				eDispencersPackageState[3].lrDoseVolumeCV 			:=3;
				eDispencersPackageState[3].bDosed					:= TRUE;				
				eDispencersPackageState[3].bDoseAborted				:= TRUE;
			END_IF
			IF NOT bDispencer4Enable THEN
				eDispencersPackageState[4].lrDoseVolumeCV 			:=3;
				eDispencersPackageState[4].bDosed					:= TRUE;				
				eDispencersPackageState[4].bDoseAborted				:= TRUE;
			END_IF
			
			
			FOR i := 1 TO 100 DO	
				
				IF eDispencersPackageState[4].nCardNumber = eRFID[i].nCardNumber AND eDispencersPackageState[4].nCardNumber > 0 THEN
					eRFID[i].lrDoseVolumeCV := ABS(lrDosedMass4CVAux);
					eRFID[i].lrDoseVolumeSV := lrDispencer1DoseVolume + VIS.lrDispencer4CorrectionWeight;
					eRFID[i].nDispencerNr := 4;
					eRFID[i].tDispencingTime := P02_Dispencers.fbDispencer4.tCycleTime;
					eRFID[i].bDosed	:=	eDispencersPackageState[4].bDosed;
					eRFID[i].bDoseAborted	:=	eDispencersPackageState[4].bDoseAborted;					
					IF NOT bDispencer4Enable THEN (*Jezeli dozowniki wylaczone to wpisz jakas wartość zeby platynki zakładało*)
						eRFID[i].lrDoseVolumeCV := 3;
					END_IF
				END_IF
							
				IF eDispencersPackageState[3].nCardNumber = eRFID[i].nCardNumber AND eDispencersPackageState[3].nCardNumber > 0 THEN
					eRFID[i].lrDoseVolumeCV := ABS(lrDosedMass3CVAux);
					eRFID[i].lrDoseVolumeSV := lrDispencer1DoseVolume + VIS.lrDispencer3CorrectionWeight;
					eRFID[i].nDispencerNr := 3;
					eRFID[i].tDispencingTime := P02_Dispencers.fbDispencer3.tCycleTime;
					eRFID[i].bDosed	:=	eDispencersPackageState[3].bDosed;
					eRFID[i].bDoseAborted	:=	eDispencersPackageState[3].bDoseAborted;	
					IF NOT bDispencer3Enable THEN (*Jezeli dozowniki wylaczone to wpisz jakas wartość zeby platynki zakładało*)
						eRFID[i].lrDoseVolumeCV := 3;
					END_IF
				END_IF
			
				IF eDispencersPackageState[2].nCardNumber = eRFID[i].nCardNumber AND eDispencersPackageState[2].nCardNumber > 0 THEN
					eRFID[i].lrDoseVolumeCV := ABS(lrDosedMass2CVAux);
					eRFID[i].lrDoseVolumeSV := lrDispencer1DoseVolume + VIS.lrDispencer2CorrectionWeight;
					eRFID[i].nDispencerNr := 2;
					eRFID[i].tDispencingTime := P02_Dispencers.fbDispencer2.tCycleTime;
					eRFID[i].bDosed	:=	eDispencersPackageState[2].bDosed;
					eRFID[i].bDoseAborted	:=	eDispencersPackageState[2].bDoseAborted;						
					IF NOT bDispencer2Enable THEN (*Jezeli dozowniki wylaczone to wpisz jakas wartość zeby platynki zakładało*)
						eRFID[i].lrDoseVolumeCV := 3;
					END_IF
				END_IF
			
				IF eDispencersPackageState[1].nCardNumber = eRFID[i].nCardNumber AND eDispencersPackageState[1].nCardNumber > 0 THEN
					eRFID[i].lrDoseVolumeCV := ABS(lrDosedMass1CVAux);
					eRFID[i].lrDoseVolumeSV := lrDispencer1DoseVolume + VIS.lrDispencer1CorrectionWeight;
					eRFID[i].nDispencerNr := 1;
					eRFID[i].tDispencingTime := P02_Dispencers.fbDispencer1.tCycleTime;
					eRFID[i].bDosed	:=	eDispencersPackageState[1].bDosed;
					eRFID[i].bDoseAborted	:=	eDispencersPackageState[1].bDoseAborted;						
					IF NOT bDispencer1Enable THEN (*Jezeli dozowniki wylaczone to wpisz jakas wartość zeby platynki zakładało*)
						eRFID[i].lrDoseVolumeCV := 3;
					END_IF
				END_IF
								
			END_FOR					
		
			IF bDispencersReadyOrSucking AND NOT (P00_PackML.fbPMLAuto.ePMLState = E_PMLState.ePMLState_STOPPING) THEN
				lrDosedMass1CVAux									:= lrDosedMass2CVAux:= 0.0;
				lrDosedMass3CVAux									:= lrDosedMass4CVAux:= 0.0;
				iDispencersCase	:=	2;
			END_IF
			
		2:
			iDispencersCase := 3;
		 
		3:	//Kasowanie sygnałów po wydozowaniu i przejscie dalej jak zniknie CycleDone
			IF NOT (P00_PackML.fbPMLAuto.ePMLState = E_PMLState.ePMLState_STOPPING) AND bDispencersReady AND bCatchersready THEN 
				VIS.bDispencer1Dose := 	VIS.bDispencer2Dose  := VIS.bDispencer3Dose  := VIS.bDispencer4Dose  := FALSE;			
				IF 	NOT P02_Dispencers.fbDispencer1.bCycleDone	AND
					NOT P02_Dispencers.fbDispencer2.bCycleDone 	AND
					NOT P02_Dispencers.fbDispencer3.bCycleDone 	AND
					NOT P02_Dispencers.fbDispencer4.bCycleDone 	AND
					NOT eDispencersPackageState[1].bDosed AND NOT eDispencersPackageState[1].bDoseAborted	AND
					NOT eDispencersPackageState[2].bDosed AND NOT eDispencersPackageState[2].bDoseAborted	AND
					NOT eDispencersPackageState[3].bDosed AND NOT eDispencersPackageState[3].bDoseAborted	AND
					NOT eDispencersPackageState[4].bDosed AND NOT eDispencersPackageState[4].bDoseAborted				
				THEN
					iDispencersCase := 4;
				END_IF
			END_IF	
			
		4:	//Dozowanie
		
			IF tonCatchDelay.Q AND NOT bChangeOver THEN	
			VIS.bDispencers1Catch 	:=	( eDispencersPackageState[1].bBottlePresent (*AND(eDispencersPackageState[1].lrDoseVolumeCV=0)*) AND bDispencersCatchEnable);
			VIS.bDispencers2Catch 	:=	( eDispencersPackageState[2].bBottlePresent (*AND(eDispencersPackageState[2].lrDoseVolumeCV=0)*) AND bDispencersCatchEnable);
			VIS.bDispencers3Catch 	:=	( eDispencersPackageState[3].bBottlePresent (*AND(eDispencersPackageState[3].lrDoseVolumeCV=0)*) AND bDispencersCatchEnable);
			VIS.bDispencers4Catch 	:=	( eDispencersPackageState[4].bBottlePresent (*AND(eDispencersPackageState[4].lrDoseVolumeCV=0)*) AND bDispencersCatchEnable);
			END_IF	
		
			IF tonDosingDelay.Q THEN		
				
				(*Wykrywanie czy jest butelka po chwyceniu chwytaka*)
				IF NOT bPhaseChanging AND NOT bChangeOver THEN //Blokada od zmiany
					VIS.bDispencer1Dose:=eDispencersPackageState[1].bBottlePresent AND (eDispencersPackageState[1].lrDoseVolumeCV=0) AND 
										(eDispencersPackageState[1].lrDoseVolumeCVSecondPhase=0) AND (fbDispencer1BottleInCatcherSensor.bOUT OR NOT bDispencersCatchEnable)
										AND NOT eDispencersPackageState[1].bDoseAborted AND bDispencer12AllowDosingAfterDrag; 
					VIS.bDispencer2Dose:=eDispencersPackageState[2].bBottlePresent AND (eDispencersPackageState[2].lrDoseVolumeCV=0) AND 
										(eDispencersPackageState[2].lrDoseVolumeCVSecondPhase=0) AND (fbDispencer2BottleInCatcherSensor.bOUT OR NOT bDispencersCatchEnable)
										AND NOT eDispencersPackageState[2].bDoseAborted AND bDispencer12AllowDosingAfterDrag; 
					VIS.bDispencer3Dose:=eDispencersPackageState[3].bBottlePresent AND (eDispencersPackageState[3].lrDoseVolumeCV=0) AND 
										(eDispencersPackageState[3].lrDoseVolumeCVSecondPhase=0) AND (fbDispencer3BottleInCatcherSensor.bOUT OR NOT bDispencersCatchEnable)
										AND NOT eDispencersPackageState[3].bDoseAborted AND bDispencer34AllowDosingAfterDrag; 										
					VIS.bDispencer4Dose:=eDispencersPackageState[4].bBottlePresent AND (eDispencersPackageState[4].lrDoseVolumeCV=0) AND 
										(eDispencersPackageState[4].lrDoseVolumeCVSecondPhase=0) AND (fbDispencer4BottleInCatcherSensor.bOUT OR NOT bDispencersCatchEnable)
										AND NOT eDispencersPackageState[4].bDoseAborted AND bDispencer34AllowDosingAfterDrag; 		
				END_IF										
				IF  ((tonbDosingDone.Q (* bDosingDone OR bDosingDoneFaster*)) AND tonDispencersCase4Delay.Q) OR
					bChangeOver
				THEN
					iDispencersCase := 1;
				END_IF	
				(*Zachowanie miedzy innymi po ESTOPIE, jeżeli coś zostało wydozowane a przerwało cykl to ustawia Aborted*)
				IF 	(ABS(lrDosedMass1CVAux) > 0 AND NOT fbDispencer1BottleInCatcherSensor.bOUT AND bDispencersCatchEnable) OR NOT fbIbDispencer12NoColisionWhenDosingSensor.bOut THEN
					eDispencersPackageState[1].bDoseAborted := TRUE;
				END_IF
				IF 	(ABS(lrDosedMass2CVAux) > 0 AND NOT fbDispencer2BottleInCatcherSensor.bOUT AND bDispencersCatchEnable) OR NOT fbIbDispencer12NoColisionWhenDosingSensor.bOut THEN
					eDispencersPackageState[2].bDoseAborted := TRUE;
				END_IF
				IF 	(ABS(lrDosedMass3CVAux) > 0 AND NOT fbDispencer3BottleInCatcherSensor.bOUT AND bDispencersCatchEnable) OR NOT fbIbDispencer34NoColisionWhenDosingSensor.bOut THEN
					eDispencersPackageState[3].bDoseAborted := TRUE;
				END_IF
				IF 	(ABS(lrDosedMass4CVAux) > 0 AND NOT fbDispencer4BottleInCatcherSensor.bOUT AND bDispencersCatchEnable) OR NOT fbIbDispencer34NoColisionWhenDosingSensor.bOut THEN
					eDispencersPackageState[4].bDoseAborted := TRUE;
				END_IF							
			END_IF
			//Szukanie ilości dozy, przeisywanie maxa i kasowanie zmienych po przepisaniu w innym cyklu
			IF P02_Dispencers.fbDispencer1.lrDosedMassCV < lrDosedMass1CVAux THEN lrDosedMass1CVAux := P02_Dispencers.fbDispencer1.lrDosedMassCV; END_IF
			IF P02_Dispencers.fbDispencer2.lrDosedMassCV < lrDosedMass2CVAux THEN lrDosedMass2CVAux := P02_Dispencers.fbDispencer2.lrDosedMassCV; END_IF
			IF P02_Dispencers.fbDispencer3.lrDosedMassCV < lrDosedMass3CVAux THEN lrDosedMass3CVAux := P02_Dispencers.fbDispencer3.lrDosedMassCV; END_IF
			IF P02_Dispencers.fbDispencer4.lrDosedMassCV < lrDosedMass4CVAux THEN lrDosedMass4CVAux := P02_Dispencers.fbDispencer4.lrDosedMassCV; END_IF
			
			IF NOT bDispencer1Enable AND NOT bDispencer2Enable AND NOT bDispencer3Enable AND NOT bDispencer4Enable
			THEN //Opcja platynkowanai jak dozowniki są wyłączone
				lrDosedMass1CVAux := lrDosedMass2CVAux := lrDosedMass3CVAux :=lrDosedMass4CVAux :=10;
			END_IF
	
	END_CASE
END_ACTION

ACTION aP02_Dispencers2Phase:
(***********************************)
(**********P02_Dispencers***********)


tonDosingDelay				(IN:=iDispencersCase=4
								,PT:=UINT_TO_TIME(uiDispencerStartDosingDelay+300));//Opoznienie przed dozowaniem //Check
tonCatchDelay				(IN:=iDispencersCase=4
								,PT:=UINT_TO_TIME(uiDispencerStartDosingDelay));//Opoznienie przed dozowaniem //Check
								
								
tonErrorDosing1					(IN:=VIS.bDispencer1Dose, PT:=T#20S);//Timer za długiego dozowania
tonErrorDosing2					(IN:=VIS.bDispencer2Dose, PT:=T#20S);
tonErrorDosing3					(IN:=VIS.bDispencer3Dose, PT:=T#20S);
tonErrorDosing4					(IN:=VIS.bDispencer4Dose, PT:=T#20S);

bDisp1FormsAndNoBottle			 := eDispencer12PackageState2Phase[1].bFormPresent AND NOT eDispencer12PackageState2Phase[1].bBottlePresent ;//Sygnały chytaków bez butelek
bDisp2FormsAndNoBottle			 := eDispencer12PackageState2Phase[2].bFormPresent AND NOT eDispencer12PackageState2Phase[2].bBottlePresent;
bDisp3FormsAndNoBottle			 := eDispencer34PackageState2Phase[1].bFormPresent AND NOT eDispencer34PackageState2Phase[1].bBottlePresent;
bDisp4FormsAndNoBottle			 := eDispencer34PackageState2Phase[2].bFormPresent AND NOT eDispencer34PackageState2Phase[2].bBottlePresent;

	tonDispencersCase4Delay(IN:=iDispencersCase=4,PT:=T#200MS); // było 100MS

//Sygnał zakończenia dozowania
bDosingDone  := 				(	NOT bDispencer1Enable OR eDispencer12PackageState2Phase[1].bDoseAbortedSecondPhase OR	
																(
																(VIS.bDispencer1Dose AND (P02_Dispencers.fbDispencer1.bCycleDone OR tonErrorDosing1.Q))  OR 
																NOT VIS.bDispencer1Dose
																)  
								)  AND 
								(	NOT bDispencer2Enable OR eDispencer12PackageState2Phase[2].bDoseAbortedSecondPhase OR 
																(
																(VIS.bDispencer2Dose AND (P02_Dispencers.fbDispencer2.bCycleDone  OR tonErrorDosing2.Q)) OR
																 NOT VIS.bDispencer2Dose
																)  
								)  AND 
								(	NOT bDispencer3Enable OR eDispencer34PackageState2Phase[1].bDoseAborted OR 
																(
																(VIS.bDispencer3Dose AND (P02_Dispencers.fbDispencer3.bCycleDone  OR tonErrorDosing3.Q)) OR
																 NOT VIS.bDispencer3Dose
																)  
								)  AND 
								(	NOT bDispencer4Enable OR eDispencer34PackageState2Phase[2].bDoseAborted OR 
																(
																(VIS.bDispencer4Dose AND (P02_Dispencers.fbDispencer4.bCycleDone  OR tonErrorDosing4.Q)) OR
																 NOT VIS.bDispencer4Dose
																)  
								)  AND 
								( iDispencersCase = 4 AND tonDosingDelay.Q) AND 
								(
									tonCatchNotEnable.Q OR tonCatched.Q OR 
									(bDisp1FormsAndNoBottle AND bDisp2FormsAndNoBottle AND bDisp3FormsAndNoBottle AND bDisp4FormsAndNoBottle) OR 
									(NOT bDispencer1Enable AND NOT bDispencer2Enable AND NOT bDispencer3Enable AND NOT bDispencer4Enable) 
								);
								
bDosingDoneFaster:=		    (tonCatched.Q AND 																											//Dorobilem bottle present
								 ((VIS.bDispencer1Dose AND P02_Dispencers.QbDispencer1DropCatcherValveActuator) OR NOT bDispencer1Enable OR NOT eDispencer12PackageState2Phase[1].bBottlePresent)
                                  AND
                                  ((VIS.bDispencer2Dose AND P02_Dispencers.QbDispencer2DropCatcherValveActuator) OR NOT bDispencer2Enable OR NOT eDispencer12PackageState2Phase[2].bBottlePresent)                                                                                               (*Dodano szybsze otwieranie szlabanu jak tylko tacki się zamkną*)                     
                                  AND
                                  ((VIS.bDispencer3Dose AND P02_Dispencers.QbDispencer3DropCatcherValveActuator) OR NOT bDispencer3Enable OR NOT eDispencer34PackageState2Phase[1].bBottlePresent)
                                  AND
                                  ((VIS.bDispencer4Dose AND P02_Dispencers.QbDispencer4DropCatcherValveActuator) OR NOT bDispencer4Enable OR NOT eDispencer34PackageState2Phase[2].bBottlePresent)                                                                                               (*Dodano szybsze otwieranie szlabanu jak tylko tacki się zamkną*)                     
                                 		  
								  
								  
                			 )
                   OR               // Dodanie jeżeli tacki się nie wysuwają to przesuwaj szybciej jeżeli dozowniki są w zasysaniu
                   (               ((VIS.bDispencer1Dose AND P02_Dispencers.fbDispencer1.eRunningState = E_DispencerState.eSucking) OR NOT bDispencer1Enable)
									 AND
									 ((VIS.bDispencer2Dose AND P02_Dispencers.fbDispencer2.eRunningState = E_DispencerState.eSucking) OR NOT bDispencer2Enable)   
									 AND
									 ((VIS.bDispencer3Dose AND P02_Dispencers.fbDispencer3.eRunningState = E_DispencerState.eSucking) OR NOT bDispencer3Enable)
									 AND
									 ((VIS.bDispencer4Dose AND P02_Dispencers.fbDispencer4.eRunningState = E_DispencerState.eSucking) OR NOT bDispencer4Enable)
                   );						
													
bDispencersReady := 			(NOT bDispencer1Enable OR P02_Dispencers.fbDispencer1.eState = E_Station.eReady) AND 
								(NOT bDispencer2Enable OR P02_Dispencers.fbDispencer2.eState = E_Station.eReady) AND	
								(NOT bDispencer3Enable OR P02_Dispencers.fbDispencer3.eState = E_Station.eReady) AND
								(NOT bDispencer4Enable OR P02_Dispencers.fbDispencer4.eState = E_Station.eReady) AND																	
								(
								NOT bDispencersCatchEnable OR (NOT bDispencer1Enable AND NOT bDispencer2Enable AND NOT bDispencer3Enable AND NOT bDispencer4Enable) OR 
								(
									(P02_Dispencers.fbDispencersCatch1Station.eState=E_Station.eReady AND NOT P02_Dispencers.fbDispencersCatch1Station.bCycleDone) AND
									(P02_Dispencers.fbDispencersCatch2Station.eState=E_Station.eReady AND NOT P02_Dispencers.fbDispencersCatch2Station.bCycleDone) AND
									(P02_Dispencers.fbDispencersCatch3Station.eState=E_Station.eReady AND NOT P02_Dispencers.fbDispencersCatch3Station.bCycleDone) AND
									(P02_Dispencers.fbDispencersCatch4Station.eState=E_Station.eReady AND NOT P02_Dispencers.fbDispencersCatch4Station.bCycleDone) 
								)
								);											
					
bDispencersReadyOrSucking := 	(NOT bDispencer1Enable OR P02_Dispencers.fbDispencer1.eState = E_Station.eReady OR P02_Dispencers.fbDispencer1.eRunningState = E_DispencerState.eSucking	OR (P02_Dispencers.fbDispencer1.eRunningState = E_DispencerState.eGoingUp	AND P02_Dispencers.QbDispencer1DropCatcherValveActuator)) AND 
								(NOT bDispencer2Enable OR P02_Dispencers.fbDispencer2.eState = E_Station.eReady OR P02_Dispencers.fbDispencer2.eRunningState = E_DispencerState.eSucking	OR (P02_Dispencers.fbDispencer2.eRunningState = E_DispencerState.eGoingUp	AND P02_Dispencers.QbDispencer2DropCatcherValveActuator)) AND
								(NOT bDispencer3Enable OR P02_Dispencers.fbDispencer3.eState = E_Station.eReady OR P02_Dispencers.fbDispencer3.eRunningState = E_DispencerState.eSucking	OR (P02_Dispencers.fbDispencer3.eRunningState = E_DispencerState.eGoingUp	AND P02_Dispencers.QbDispencer3DropCatcherValveActuator)) AND
								(NOT bDispencer4Enable OR P02_Dispencers.fbDispencer4.eState = E_Station.eReady OR P02_Dispencers.fbDispencer4.eRunningState = E_DispencerState.eSucking	OR (P02_Dispencers.fbDispencer4.eRunningState = E_DispencerState.eGoingUp	AND P02_Dispencers.QbDispencer4DropCatcherValveActuator));
bCatchersReady:=		NOT bDispencersCatchEnable OR (NOT bDispencer1Enable AND NOT bDispencer2Enable AND NOT bDispencer3Enable AND NOT bDispencer4Enable) OR 
								(
									(P02_Dispencers.fbDispencersCatch1Station.eState=E_Station.eReady AND NOT P02_Dispencers.fbDispencersCatch1Station.bCycleDone) AND
									(P02_Dispencers.fbDispencersCatch2Station.eState=E_Station.eReady AND NOT P02_Dispencers.fbDispencersCatch2Station.bCycleDone) AND
									(P02_Dispencers.fbDispencersCatch3Station.eState=E_Station.eReady AND NOT P02_Dispencers.fbDispencersCatch3Station.bCycleDone) AND
									(P02_Dispencers.fbDispencersCatch4Station.eState=E_Station.eReady AND NOT P02_Dispencers.fbDispencersCatch4Station.bCycleDone) 
								)			;
																
//Timer braku chwytania opakowania
tonCatchNotEnable				(IN:=NOT bDispencersCatchEnable AND 
								(
									VIS.bDispencer1Dose OR VIS.bDispencer2Dose OR VIS.bDispencer3Dose OR VIS.bDispencer4Dose OR 
									(
									(P02_Dispencers.fbDispencer1.eRunningState = E_DispencerState.eSucking OR NOT bDispencer1Enable) OR 
									(P02_Dispencers.fbDispencer2.eRunningState = E_DispencerState.eSucking OR NOT bDispencer2Enable) OR
									(P02_Dispencers.fbDispencer3.eRunningState = E_DispencerState.eSucking OR NOT bDispencer3Enable) OR 
									(P02_Dispencers.fbDispencer4.eRunningState = E_DispencerState.eSucking OR NOT bDispencer4Enable) 
									)
								),PT:=T#20MS);
//Opoznienie chwycenia
tonCatched						(IN:=	(P02_Dispencers.fbDispencersCatch1Station.eRunningState=E_CatchStationState.eCatched OR P02_Dispencers.fbDispencersCatch1Station.eRunningState=E_CatchStationState.eNotCatched OR  NOT eDispencer12PackageState2Phase[1].bBottlePresent OR NOT bDispencer1Enable) AND
										(P02_Dispencers.fbDispencersCatch2Station.eRunningState=E_CatchStationState.eCatched OR P02_Dispencers.fbDispencersCatch2Station.eRunningState=E_CatchStationState.eNotCatched OR  NOT eDispencer12PackageState2Phase[2].bBottlePresent OR NOT bDispencer2Enable) AND
										(P02_Dispencers.fbDispencersCatch3Station.eRunningState=E_CatchStationState.eCatched OR P02_Dispencers.fbDispencersCatch3Station.eRunningState=E_CatchStationState.eNotCatched OR  NOT eDispencer34PackageState2Phase[1].bBottlePresent OR NOT bDispencer3Enable) AND
										(P02_Dispencers.fbDispencersCatch4Station.eRunningState=E_CatchStationState.eCatched OR P02_Dispencers.fbDispencersCatch4Station.eRunningState=E_CatchStationState.eNotCatched OR  NOT eDispencer34PackageState2Phase[2].bBottlePresent OR NOT bDispencer4Enable)
										,PT:=T#500MS);
										
//Filtry sygnałów wykrywania butelek pod chwytakiem
bDispencer1CatchedOrNoBottle := P02_Dispencers.fbDispencersCatch1Station.eRunningState=E_CatchStationState.eCatched OR NOT eDispencer12PackageState2Phase[1].bBottlePresent;
bDispencer2CatchedOrNoBottle := P02_Dispencers.fbDispencersCatch2Station.eRunningState=E_CatchStationState.eCatched OR NOT eDispencer12PackageState2Phase[2].bBottlePresent;
bDispencer3CatchedOrNoBottle := P02_Dispencers.fbDispencersCatch3Station.eRunningState=E_CatchStationState.eCatched OR NOT eDispencer34PackageState2Phase[1].bBottlePresent;
bDispencer4CatchedOrNoBottle := P02_Dispencers.fbDispencersCatch4Station.eRunningState=E_CatchStationState.eCatched OR NOT eDispencer34PackageState2Phase[2].bBottlePresent;

fbDispencer1BottleInCatcherSensor(bIN:=P02_Dispencers.fbDispencersCatch1Station.eRunningState=E_CatchStationState.eCatched AND bDispencer2CatchedOrNoBottle AND IbEmergencyStop, tFilterTimeOn:=T#50MS, tFilterTimeOff:=T#100MS, bOUT=> );(*Filtr wejścia cyfrowego*)
fbDispencer2BottleInCatcherSensor(bIN:=P02_Dispencers.fbDispencersCatch2Station.eRunningState=E_CatchStationState.eCatched AND bDispencer1CatchedOrNoBottle AND IbEmergencyStop, tFilterTimeOn:=T#50MS, tFilterTimeOff:=T#100MS, bOUT=> );(*Filtr wejścia cyfrowego*)//bylo 150
fbDispencer3BottleInCatcherSensor(bIN:=P02_Dispencers.fbDispencersCatch3Station.eRunningState=E_CatchStationState.eCatched AND bDispencer4CatchedOrNoBottle AND IbEmergencyStop, tFilterTimeOn:=T#50MS, tFilterTimeOff:=T#100MS, bOUT=> );(*Filtr wejścia cyfrowego*)
fbDispencer4BottleInCatcherSensor(bIN:=P02_Dispencers.fbDispencersCatch4Station.eRunningState=E_CatchStationState.eCatched AND bDispencer3CatchedOrNoBottle AND IbEmergencyStop, tFilterTimeOn:=T#50MS, tFilterTimeOff:=T#500MS, bOUT=> );(*Filtr wejścia cyfrowego*)

CASE iDispencersCase OF

		0: //Kilka stanów niepotrzebnych, zeby zgadzało się z innymi liniami, w razie poprawek, aktualizacji
			iDispencersCase := 4;
			
		1:	//Przepisywanie danych po wydozowaniu
			
			VIS.bDispencers1Catch 	:=FALSE;
			VIS.bDispencers2Catch 	:=FALSE;
			VIS.bDispencers3Catch 	:=FALSE;
			VIS.bDispencers4Catch 	:=FALSE;
			
			(**PRZEPISYWANIE PARAMETRÓW PO WYDOZOWANIU**)
			eDispencer34PackageState2Phase[1].lrDoseVolumeCV					:= ABS(lrDosedMass3CVAux);
			eDispencer34PackageState2Phase[1].lrDoseVolumeSV 					:= lrDispencer2DoseVolume + VIS.lrDispencer3CorrectionWeight;
			eDispencer34PackageState2Phase[1].nDispencerNr 						:= 3;
			eDispencer34PackageState2Phase[1].tDispencingTime 					:= P02_Dispencers.fbDispencer3.tCycleTime;
			eDispencer34PackageState2Phase[2].lrDoseVolumeCV					:= ABS(lrDosedMass4CVAux);
			eDispencer34PackageState2Phase[2].lrDoseVolumeSV 					:= lrDispencer2DoseVolume + VIS.lrDispencer4CorrectionWeight;
			eDispencer34PackageState2Phase[2].nDispencerNr 						:= 4;
			eDispencer34PackageState2Phase[2].tDispencingTime 					:= P02_Dispencers.fbDispencer4.tCycleTime;
			
			IF NOT vis.bWeight1EnableShow THEN
			eDispencer34PackageState2Phase[1].bWeightOK							:= TRUE;
			eDispencer34PackageState2Phase[2].bWeightOK							:= TRUE;
			eDispencer12PackageState2Phase[1].bWeightOK							:= TRUE;
			eDispencer12PackageState2Phase[2].bWeightOK							:= TRUE;
			END_IF


												
			eDispencer12PackageState2Phase[1].lrDoseVolumeCVSecondPhase := ABS(lrDosedMass1CVAux);
			eDispencer12PackageState2Phase[1].lrDoseVolumeSVSecondPhase := lrDispencer1DoseVolume + VIS.lrDispencer1CorrectionWeight;
			eDispencer12PackageState2Phase[1].nDispencerNrSecondPhase := 1;
			eDispencer12PackageState2Phase[1].tDispencingTimeSecondPhase := P02_Dispencers.fbDispencer1.tCycleTime;
			eDispencer12PackageState2Phase[2].lrDoseVolumeCVSecondPhase := ABS(lrDosedMass2CVAux);
			eDispencer12PackageState2Phase[2].lrDoseVolumeSVSecondPhase := lrDispencer1DoseVolume + VIS.lrDispencer2CorrectionWeight;
			eDispencer12PackageState2Phase[2].nDispencerNrSecondPhase := 2;
			eDispencer12PackageState2Phase[2].tDispencingTimeSecondPhase := P02_Dispencers.fbDispencer2.tCycleTime;







			(*Sprawdzanie czy wydozowana ilość zgadza się z zadaną*)
			IF 	ABS(eDispencer12PackageState2Phase[1].lrDoseVolumeSVSecondPhase  - eDispencer12PackageState2Phase[1].lrDoseVolumeCVSecondPhase) < 15 // bylo >5 
				AND eDispencer12PackageState2Phase[1].bBottlePresent	THEN 
					eDispencer12PackageState2Phase[1].bDosedSecondPhase			:= TRUE;	ELSE
					eDispencer12PackageState2Phase[1].bDoseAbortedSecondPhase 	:= TRUE;	
			END_IF
			IF 	ABS(eDispencer12PackageState2Phase[2].lrDoseVolumeSVSecondPhase  - eDispencer12PackageState2Phase[2].lrDoseVolumeCVSecondPhase) < 15
				AND eDispencer12PackageState2Phase[2].bBottlePresent	THEN 
					eDispencer12PackageState2Phase[2].bDosedSecondPhase 		:= TRUE;	ELSE
					eDispencer12PackageState2Phase[2].bDoseAbortedSecondPhase 	:= TRUE;	
			END_IF
			IF 	ABS(eDispencer34PackageState2Phase[1].lrDoseVolumeSV  - eDispencer34PackageState2Phase[1].lrDoseVolumeCV) < 15
				AND eDispencer34PackageState2Phase[1].bBottlePresent	THEN 
					eDispencer34PackageState2Phase[1].bDosed := TRUE;	ELSE
					eDispencer34PackageState2Phase[1].bDoseAborted := TRUE;	
			END_IF
			IF 	ABS(eDispencer34PackageState2Phase[2].lrDoseVolumeSV  - eDispencer34PackageState2Phase[2].lrDoseVolumeCV) < 15
				AND eDispencer34PackageState2Phase[2].bBottlePresent	THEN 
					eDispencer34PackageState2Phase[2].bDosed := TRUE;	ELSE
					eDispencer34PackageState2Phase[2].bDoseAborted := TRUE;	
			END_IF

			IF NOT bDispencer1Enable THEN (*Jezeli dozowniki wylaczone to wpisz jakas wartość zeby platynki zakładało*)
				eDispencer12PackageState2Phase[1].lrDoseVolumeCVSecondPhase 			:=3;
				eDispencer12PackageState2Phase[1].bDoseAbortedSecondPhase				:= TRUE;
			END_IF
			IF NOT bDispencer2Enable THEN (*Jezeli dozowniki wylaczone to wpisz jakas wartość zeby platynki zakładało*)	
				eDispencer12PackageState2Phase[2].lrDoseVolumeCVSecondPhase  			:=3;
				eDispencer12PackageState2Phase[2].bDoseAbortedSecondPhase				:= TRUE;
			END_IF
			IF NOT bDispencer3Enable THEN (*Jezeli dozowniki wylaczone to wpisz jakas wartość zeby platynki zakładało*)
				eDispencer34PackageState2Phase[1].lrDoseVolumeCV 			:=3;
				eDispencer34PackageState2Phase[1].bDoseAborted				:= TRUE;
			END_IF
			IF NOT bDispencer4Enable THEN
				eDispencer34PackageState2Phase[2].lrDoseVolumeCV 			:=3;
				eDispencer34PackageState2Phase[2].bDoseAborted				:= TRUE;
			END_IF
			
			FOR i := 1 TO 100 DO	
				
				IF eDispencer34PackageState2Phase[2].nCardNumber = eRFID[i].nCardNumber AND eDispencer34PackageState2Phase[2].nCardNumber > 0 THEN
					//nd:=i; //Do testów
					eRFID[i].lrDoseVolumeCV := ABS(lrDosedMass4CVAux);
					eRFID[i].lrDoseVolumeSV := lrDispencer2DoseVolume + VIS.lrDispencer4CorrectionWeight;
					eRFID[i].nDispencerNr := 4;
					eRFID[i].tDispencingTime := P02_Dispencers.fbDispencer4.tCycleTime;
					eRFID[i].bDosed	:=	eDispencer34PackageState2Phase[2].bDosed;
					eRFID[i].bDoseAborted	:=	eDispencer34PackageState2Phase[2].bDoseAborted;
					eRFID[i].bWeightOK	:= eDispencer34PackageState2Phase[2].bWeightOK;
					IF NOT bDispencer4Enable THEN (*Jezeli dozowniki wylaczone to wpisz jakas wartość zeby platynki zakładało*)
						eRFID[i].lrDoseVolumeCV := 3;
					END_IF
				END_IF
							
				IF eDispencer34PackageState2Phase[1].nCardNumber = eRFID[i].nCardNumber AND eDispencer34PackageState2Phase[1].nCardNumber > 0 THEN
				//	nd:=i; //Do testów
					eRFID[i].lrDoseVolumeCV := ABS(lrDosedMass3CVAux);
					eRFID[i].lrDoseVolumeSV := lrDispencer2DoseVolume + VIS.lrDispencer3CorrectionWeight;
					eRFID[i].nDispencerNr := 3;
					eRFID[i].tDispencingTime := P02_Dispencers.fbDispencer3.tCycleTime;
					eRFID[i].bDosed	:=	eDispencer34PackageState2Phase[1].bDosed;
					eRFID[i].bDoseAborted	:=	eDispencer34PackageState2Phase[1].bDoseAborted;	
					eRFID[i].bWeightOK	:= eDispencer34PackageState2Phase[1].bWeightOK;	
					IF NOT bDispencer3Enable THEN (*Jezeli dozowniki wylaczone to wpisz jakas wartość zeby platynki zakładało*)
						eRFID[i].lrDoseVolumeCV := 3;
					END_IF
				END_IF
			
				IF eDispencer12PackageState2Phase[2].nCardNumber = eRFID[i].nCardNumber AND eDispencer12PackageState2Phase[2].nCardNumber > 0THEN
				//	nd:=i; //Do testów
					eRFID[i].lrDoseVolumeCVSecondPhase := ABS(lrDosedMass2CVAux);
					eRFID[i].lrDoseVolumeSVSecondPhase := lrDispencer1DoseVolume + VIS.lrDispencer2CorrectionWeight;
					eRFID[i].nDispencerNrSecondPhase := 2;
					eRFID[i].tDispencingTimeSecondPhase := P02_Dispencers.fbDispencer2.tCycleTime;
					eRFID[i].bDosed	:=	eDispencer12PackageState2Phase[2].bDosed;
					eRFID[i].bDoseAborted	:=	eDispencer12PackageState2Phase[2].bDoseAborted;
					eRFID[i].bWeightOK	:= eDispencer12PackageState2Phase[2].bWeightOK;		
					IF NOT bDispencer2Enable THEN (*Jezeli dozowniki wylaczone to wpisz jakas wartość zeby platynki zakładało*)
						eRFID[i].lrDoseVolumeCVSecondPhase := 3;
					END_IF
				END_IF
			
				IF eDispencer12PackageState2Phase[1].nCardNumber = eRFID[i].nCardNumber AND eDispencer12PackageState2Phase[1].nCardNumber > 0 THEN
				//	nd:=i; //Do testów
					eRFID[i].lrDoseVolumeCVSecondPhase := ABS(lrDosedMass1CVAux);
					eRFID[i].lrDoseVolumeSVSecondPhase := lrDispencer1DoseVolume + VIS.lrDispencer1CorrectionWeight;
					eRFID[i].nDispencerNrSecondPhase := 1;
					eRFID[i].tDispencingTimeSecondPhase := P02_Dispencers.fbDispencer1.tCycleTime;
					eRFID[i].bDosed	:=	eDispencer12PackageState2Phase[1].bDosed;
					eRFID[i].bDoseAborted	:=	eDispencer12PackageState2Phase[1].bDoseAborted;
					eRFID[i].bWeightOK	:= eDispencer12PackageState2Phase[1].bWeightOK;			
					IF NOT bDispencer1Enable THEN (*Jezeli dozowniki wylaczone to wpisz jakas wartość zeby platynki zakładało*)
						eRFID[i].lrDoseVolumeCVSecondPhase := 3;
					END_IF
				END_IF
								
			END_FOR	
			
			IF bDispencersReadyOrSucking AND NOT (P00_PackML.fbPMLAuto.ePMLState = E_PMLState.ePMLState_STOPPING) THEN
				lrDosedMass1CVAux									:= lrDosedMass2CVAux:= 0.0;
				lrDosedMass3CVAux									:= lrDosedMass4CVAux:= 0.0;
				iDispencersCase	:=	2;
			END_IF
			
		2:
			iDispencersCase := 3;
		 
		3:	//Kasowanie sygnałów po wydozowaniu i przejscie dalej jak zniknie CycleDone
			IF NOT (P00_PackML.fbPMLAuto.ePMLState = E_PMLState.ePMLState_STOPPING) AND bDispencersReady AND bCatchersready THEN 
				VIS.bDispencer1Dose := 	VIS.bDispencer2Dose  := VIS.bDispencer3Dose  := VIS.bDispencer4Dose  := FALSE;			
				IF 	NOT P02_Dispencers.fbDispencer1.bCycleDone	AND
					NOT P02_Dispencers.fbDispencer2.bCycleDone 	AND
					NOT P02_Dispencers.fbDispencer3.bCycleDone 	AND
					NOT P02_Dispencers.fbDispencer4.bCycleDone 	AND
					NOT eDispencer12PackageState2Phase[1].bDosedSecondPhase AND NOT eDispencer12PackageState2Phase[1].bDoseAbortedSecondPhase	AND 
					NOT eDispencer12PackageState2Phase[2].bDosedSecondPhase AND NOT eDispencer12PackageState2Phase[2].bDoseAbortedSecondPhase	AND
					NOT eDispencer34PackageState2Phase[1].bDosed AND NOT eDispencer34PackageState2Phase[1].bDoseAborted	AND
					NOT eDispencer34PackageState2Phase[2].bDosed AND NOT eDispencer34PackageState2Phase[2].bDoseAborted				
				THEN
					iDispencersCase := 4;
				END_IF
			END_IF	
			
		4:	//Dozowanie
		
			IF tonCatchDelay.Q THEN	
			VIS.bDispencers1Catch 	:=	( eDispencer12PackageState2Phase[1].bBottlePresent (*AND(eDispencersPackageState[1].lrDoseVolumeCV=0)*) AND bDispencersCatchEnable);
			VIS.bDispencers2Catch 	:=	( eDispencer12PackageState2Phase[2].bBottlePresent (*AND(eDispencersPackageState[2].lrDoseVolumeCV=0)*) AND bDispencersCatchEnable);
			VIS.bDispencers3Catch 	:=	( eDispencer34PackageState2Phase[1].bBottlePresent (*AND(eDispencersPackageState[3].lrDoseVolumeCV=0)*) AND bDispencersCatchEnable);
			VIS.bDispencers4Catch 	:=	( eDispencer34PackageState2Phase[2].bBottlePresent (*AND(eDispencersPackageState[4].lrDoseVolumeCV=0)*) AND bDispencersCatchEnable);
			END_IF	
		
			IF tonDosingDelay.Q THEN		
				IF NOT bPhaseChanging THEN //Blokada od zmiany				
					(*Wykrywanie czy jest butelka po chwyceniu chwytaka*)
					VIS.bDispencer1Dose:=eDispencer12PackageState2Phase[1].bBottlePresent AND 
										(eDispencer12PackageState2Phase[1].lrDoseVolumeCVSecondPhase=0) AND (fbDispencer1BottleInCatcherSensor.bOUT OR NOT bDispencersCatchEnable)
										AND NOT eDispencer12PackageState2Phase[1].bDoseAbortedSecondPhase; 
					VIS.bDispencer2Dose:=eDispencer12PackageState2Phase[2].bBottlePresent AND 
										(eDispencer12PackageState2Phase[2].lrDoseVolumeCVSecondPhase=0) AND (fbDispencer2BottleInCatcherSensor.bOUT OR NOT bDispencersCatchEnable)
										AND NOT eDispencersPackageState[2].bDoseAbortedSecondPhase; 
					VIS.bDispencer3Dose:=eDispencer34PackageState2Phase[1].bBottlePresent AND (eDispencer34PackageState2Phase[1].lrDoseVolumeCV=0) AND 
										(eDispencer34PackageState2Phase[1].lrDoseVolumeCVSecondPhase=0) AND (fbDispencer3BottleInCatcherSensor.bOUT OR NOT bDispencersCatchEnable)
										AND NOT eDispencer34PackageState2Phase[1].bDoseAborted; 										
					VIS.bDispencer4Dose:=eDispencer34PackageState2Phase[2].bBottlePresent AND (eDispencer34PackageState2Phase[2].lrDoseVolumeCV=0) AND 
										(eDispencer34PackageState2Phase[2].lrDoseVolumeCVSecondPhase=0) AND (fbDispencer4BottleInCatcherSensor.bOUT OR NOT bDispencersCatchEnable)
										AND NOT eDispencer34PackageState2Phase[2].bDoseAborted; 		
				END_IF								
				IF  (bDosingDone OR bDosingDoneFaster) AND tonDispencersCase4Delay.Q	THEN
					iDispencersCase := 1;
				END_IF	
					
				(*Zachowanie miedzy innymi po ESTOPIE, jeżeli coś zostało wydozowane a przerwało cykl to ustawia Aborted*)
				IF 	(ABS(lrDosedMass1CVAux) > 0 AND NOT fbDispencer1BottleInCatcherSensor.bOUT AND bDispencersCatchEnable) OR NOT fbIbDispencer12NoColisionWhenDosingSensor.bOut THEN
					eDispencer12PackageState2Phase[1].bDoseAbortedSecondPhase := TRUE;
				END_IF
				IF 	(ABS(lrDosedMass2CVAux) > 0 AND NOT fbDispencer2BottleInCatcherSensor.bOUT AND bDispencersCatchEnable) OR NOT fbIbDispencer12NoColisionWhenDosingSensor.bOut THEN
					eDispencer12PackageState2Phase[2].bDoseAbortedSecondPhase := TRUE;
				END_IF
				IF 	(ABS(lrDosedMass3CVAux) > 0 AND NOT fbDispencer3BottleInCatcherSensor.bOUT AND bDispencersCatchEnable) OR NOT fbIbDispencer34NoColisionWhenDosingSensor.bOut THEN
					eDispencer34PackageState2Phase[1].bDoseAborted := TRUE;
				END_IF
				IF 	(ABS(lrDosedMass4CVAux) > 0 AND NOT fbDispencer4BottleInCatcherSensor.bOUT AND bDispencersCatchEnable) OR NOT fbIbDispencer34NoColisionWhenDosingSensor.bOut THEN
					eDispencer34PackageState2Phase[2].bDoseAborted := TRUE;
				END_IF				
			
			END_IF
			//Szukanie ilości dozy, przeisywanie maxa i kasowanie zmienych po przepisaniu w innym cyklu
			IF P02_Dispencers.fbDispencer1.lrDosedMassCV < lrDosedMass1CVAux THEN lrDosedMass1CVAux := P02_Dispencers.fbDispencer1.lrDosedMassCV; END_IF
			IF P02_Dispencers.fbDispencer2.lrDosedMassCV < lrDosedMass2CVAux THEN lrDosedMass2CVAux := P02_Dispencers.fbDispencer2.lrDosedMassCV; END_IF
			IF P02_Dispencers.fbDispencer3.lrDosedMassCV < lrDosedMass3CVAux THEN lrDosedMass3CVAux := P02_Dispencers.fbDispencer3.lrDosedMassCV; END_IF
			IF P02_Dispencers.fbDispencer4.lrDosedMassCV < lrDosedMass4CVAux THEN lrDosedMass4CVAux := P02_Dispencers.fbDispencer4.lrDosedMassCV; END_IF
			
			IF NOT bDispencer1Enable AND NOT bDispencer2Enable AND NOT bDispencer3Enable AND NOT bDispencer4Enable THEN //Opcja platynkowanai jak dozowniki są wyłączone
				lrDosedMass1CVAux := lrDosedMass2CVAux := lrDosedMass3CVAux :=lrDosedMass4CVAux :=10;
			END_IF
	
	END_CASE
END_ACTION

ACTION aP02_Drag1Phase_GateAfter:
//Reset zmiennych jeśli mamy Stopping
IF P00_PackML.fbPMLAuto.ePMLState = E_PMLState.ePMLState_STOPPING THEN
	GVL.bFormsDragingRightPrepareRun							:= FALSE;
	VIS.bFormsDragingRightRun									:= FALSE;
	GVL.bFormsDragingLeftPrepareRun								:= FALSE;
	VIS.bFormsDragingLeftRun									:= FALSE;
		bFormsDragingRightRunCheck								:= FALSE;
		bFormsDragingLeftRunCheck								:= FALSE;	
END_IF

//Liczenie formatek
iFormatOnWeightCounter:= BOOL_TO_UINT(eWeightPackageState[1].bFormPresent) + BOOL_TO_UINT(eWeightPackageState[2].bFormPresent) + BOOL_TO_UINT(eWeightPackageState[3].bFormPresent) +
 						 BOOL_TO_UINT(eWeightPackageState[4].bFormPresent) + BOOL_TO_UINT(eWeightPackageState[5].bFormPresent);


(*** ROZPOCZECIE KONFEKCJI PO RESECIE CYKLU***)
// Wykonanie jednego przeciągania, żeby pozbyć się formatek spod dozowników
IF (P00_PackML.rtLongDelayFirstDraging.Q OR brtLongDelayFirstDraging) AND NOT bPhaseChanging AND NOT fbIbDispencerAfterCheckFormSensor.bOut THEN
	brtLongDelayFirstDraging									:=	TRUE;
	brtLongDelayFirstDragingDone								:=	TRUE;	
	IF tonFourthFormatSensor.Q THEN
		brtLongDelayFirstDraging								:= FALSE;
		bFormsDragingRightRunCheck								:= TRUE;
		bFormsDragingLeftRunCheck								:= TRUE;
		//VIS.bFormsDragingRightRun								:= TRUE;
		//VIS.bFormsDragingLeftRun								:= TRUE; 
		iTestDrag:=iTestDrag+1;
	END_IF
	IF P02_Dispencers.fbDispencersDragRightStation.bCycleDone AND  P02_Dispencers.fbDispencersDragLeftStation.bCycleDone THEN
		VIS.bFormsDragingRightRun								:= FALSE;
		GVL.bFormsDragingRightPrepareRun						:= FALSE;
		VIS.bFormsDragingLeftRun								:= FALSE;
		GVL.bFormsDragingLeftPrepareRun							:= FALSE;
		brtLongDelayFirstDraging								:= FALSE;
		bFormsDragingRightRunCheck								:= FALSE;
		bFormsDragingLeftRunCheck								:= FALSE;			
	END_IF
END_IF

// Licz. formatek przed dozownikami
tonFormsDragingFormCounter4		(IN:=iFormsDragingFormCounter <> 4	AND Main.IbFourthFormCheckFormSensor,	PT:=T#10S);
tonFormsDragingFormCounter4b	(IN:=iFormsDragingFormCounter > 4	AND Main.IbFourthFormCheckFormSensor,	PT:=T#10S);
tonCapSorterDragFormCounter4.ET;
IF tonFormsDragingFormCounter4.Q THEN
	iFormsDragingFormCounter		:=	4;
	itonFormsDragingFormCounter4	:=	itonFormsDragingFormCounter4	+	1;
END_IF
IF tonFormsDragingFormCounter4b.Q THEN
	iFormsDragingFormCounter		:=	4;
	itonFormsDragingFormCounter4b	:=	itonFormsDragingFormCounter4b	+	1;	
END_IF
IF 	P02_Dispencers.eDispencersDragLeftRunningStation = E_DragStationState.eDraging AND NOT Main.IbFourthFormCheckFormSensor AND NOT MAIN.IbSecondFormCheckFormSensor THEN
	iFormsDragingFormCounter		:= 0;
END_IF
// Koniec Licz. formatek przed dozownikami

bCatchersReady2	:=	NOT bDispencersCatchEnable OR (NOT bDispencer1Enable AND NOT bDispencer2Enable AND NOT bDispencer3Enable AND NOT bDispencer4Enable) OR 
							(
								(P02_Dispencers.fbDispencersCatch1Station.eState=E_Station.eReady AND NOT P02_Dispencers.fbDispencersCatch1Station.bCycleDone) AND
								(P02_Dispencers.fbDispencersCatch2Station.eState=E_Station.eReady AND NOT P02_Dispencers.fbDispencersCatch2Station.bCycleDone) AND
								(P02_Dispencers.fbDispencersCatch3Station.eState=E_Station.eReady AND NOT P02_Dispencers.fbDispencersCatch3Station.bCycleDone) AND
								(P02_Dispencers.fbDispencersCatch4Station.eState=E_Station.eReady AND NOT P02_Dispencers.fbDispencersCatch4Station.bCycleDone) 
							)			;

IF tonDelayAfterStart6s.Q AND NOT brtLongDelayFirstDraging AND NOT (iGateDispCase=200) AND NOT bPhaseChanging THEN //Czas po którym możemy przejść do cyklu i brak ropoczęcia konfekcji
	
	//Mamy 4 Formatki w rejestrze przed Dozownikami
	IF 
	 	tonLongDelayAfterStart.Q	AND
		eBeforeDispencersPackageState[1].bFormPresent AND eBeforeDispencersPackageState[2].bFormPresent AND 
	   	eBeforeDispencersPackageState[3].bFormPresent AND eBeforeDispencersPackageState[4].bFormPresent AND 
		NOT P02_Dispencers.fbDispencersDragRightStation.bCycleDone AND NOT P02_Dispencers.fbDispencersDragLeftStation.bCycleDone THEN
		
	   	//4 Formatka stoi na czujniku prze czas T
		IF tonFourthFormatSensor.Q AND NOT (P00_PackML.fbPMLAuto.ePMLState = E_PMLState.ePMLState_STOPPING) THEN
			GVL.bFormsDragingRightPrepareRun							:= TRUE;
			GVL.bFormsDragingLeftPrepareRun								:= TRUE;
		END_IF
	
		//Dozowniki wykonały cykl lub nie było butelki
		IF ((eDispencersPackageState[1].bFormPresent AND eDispencersPackageState[1].bBottlePresent AND (eDispencersPackageState[1].bDosed OR  eDispencersPackageState[1].bDoseAborted)) OR NOT eDispencersPackageState[1].bBottlePresent) AND
		   ((eDispencersPackageState[2].bFormPresent AND eDispencersPackageState[2].bBottlePresent AND (eDispencersPackageState[2].bDosed OR  eDispencersPackageState[2].bDoseAborted)) OR NOT eDispencersPackageState[2].bBottlePresent) AND
		   ((eDispencersPackageState[3].bFormPresent AND eDispencersPackageState[3].bBottlePresent AND (eDispencersPackageState[3].bDosed OR  eDispencersPackageState[3].bDoseAborted)) OR NOT eDispencersPackageState[3].bBottlePresent) AND
		   ((eDispencersPackageState[4].bFormPresent AND eDispencersPackageState[4].bBottlePresent AND (eDispencersPackageState[4].bDosed OR  eDispencersPackageState[4].bDoseAborted)) OR NOT eDispencersPackageState[4].bBottlePresent) THEN
		
		   	//Rejest za dozownikamu pusty i możemy przeciągać
			IF NOT eAfterDispencersPackageState[1].bFormPresent AND NOT eAfterDispencersPackageState[2].bFormPresent AND NOT eAfterDispencersPackageState[3].bFormPresent AND NOT eAfterDispencersPackageState[4].bFormPresent AND
				NOT (P05_Weight.eWeightStationRunningState = E_WeightLiftStationState.eRepair) AND NOT 
				MAIN.IbTwoPhasesFormSensorBetweenDispencers AND 
				NOT fbIbDispencerAfterCheckFormSensor.bOut	AND	
				//NOT P05_Weight.fbIbWeight4FormBeforeSensor.bOut 
				//iFormsDragingFormCounter = 4 AND
//				fbIbWeight14Gate4FormBeforeSensor.bOut
				(fbIbWeight14Gate4FormBeforeSensor.bOut OR (VIS.bGateBeforeWeight14Run AND P01_Gates.IbGateBeforeWeights14Sensor))
				
			THEN
			
				IF nFormTransportersBeforeScrewerVelocitySV < 610 THEN
					IF P01_Gates.QbGateBeforeDispencersActuator  AND tonFourthFormatSensor.Q AND bCatchersReady2 AND 
	//				(VIS.iNumbersOfFormsBetweenWeightAndScrewers <= P00_PackML.iSetNumbersOfFormsBetweenWeightAndScrewers OR VIS.bWeight1EnableShow)
					(NOT fbIbCapSorterGateWeightSensor.bOUT OR VIS.bWeight1EnableShow) // dp ZL
					AND (tonFourthFormatSensor2.Q OR NOT bCapSorterDragIfNot4PucksAnd5sRepair)
					THEN // zmieniona ilośc na 2 a było 3 formatki
						bCapSorterDragIfNot4PucksAnd5sRepair	:= FALSE;
						//VIS.bFormsDragingLeftRun				:= TRUE; 
						bFormsDragingRightRunCheck				:= TRUE; 
						bFormsDragingLeftRunCheck				:= TRUE; 	
					END_IF
				ELSE
					IF P01_Gates.QbGateBeforeDispencersActuator AND tonFourthFormatSensor.Q AND bCatchersReady2 AND 
	//				(VIS.iNumbersOfFormsBetweenWeightAndScrewers <= P00_PackML.iSetNumbersOfFormsBetweenWeightAndScrewers OR VIS.bWeight1EnableShow)
					(NOT fbIbCapSorterGateWeightSensor.bOUT OR VIS.bWeight1EnableShow) // dp ZL
					AND (tonFourthFormatSensor2.Q OR NOT bCapSorterDragIfNot4PucksAnd5sRepair)
					THEN // zmieniona ilośc na 2 a było 3 formatki
						bCapSorterDragIfNot4PucksAnd5sRepair	:= FALSE;
						bFormsDragingRightRunCheck				:= TRUE; 						
						bFormsDragingLeftRunCheck				:= TRUE; 
					END_IF
				END_IF
				
			END_IF 
		END_IF  
	END_IF	
	
	//CycleDone, resetuje pozwolenia
	IF P02_Dispencers.fbDispencersDragRightStation.bCycleDone THEN
		VIS.bFormsDragingRightRun								:= FALSE;
		GVL.bFormsDragingRightPrepareRun						:= FALSE;
		bFormsDragingRightRunCheck								:= FALSE;
	END_IF
	
	//CycleDone, resetuje pozwolenia
	IF P02_Dispencers.fbDispencersDragLeftStation.bCycleDone THEN
		VIS.bFormsDragingLeftRun								:= FALSE;
		GVL.bFormsDragingLeftPrepareRun							:= FALSE;
		bFormsDragingLeftRunCheck								:= FALSE;		
	END_IF
	
END_IF
END_ACTION

ACTION aP02_Drag2Phase_GateAfter:
//Reset zmiennych jeśli mamy Stopping
IF P00_PackML.fbPMLAuto.ePMLState = E_PMLState.ePMLState_STOPPING THEN
	GVL.bFormsDragingRightPrepareRun							:= FALSE;
	VIS.bFormsDragingRightRun									:= FALSE;
	GVL.bFormsDragingLeftPrepareRun								:= FALSE;
	VIS.bFormsDragingLeftRun									:= FALSE;
	bFormsDragingLeftRunCheck									:= FALSE;			
	bFormsDragingRightRunCheck									:= FALSE;		
END_IF

tofWeight6FormSensor	(IN:=P05_Weight.IbWeight6FormSensor, PT:=T#600MS);
tofbacktodrag			(IN:=tonQueAfterPlatin.q, PT:=T#4S);
tofQueAfterPlatinForDisp (IN:=tonQueAfterPlatin.q, PT:=T#5S);
tonQueBeforePlatins	(IN:=MAIN.IbLidFeederAfterSensor, PT:=T#3S);
//Liczenie formatek
iFormatOnWeight2PhaseCounter:= BOOL_TO_UINT(eWeightPackage2PhasePackageState[1].bFormPresent) + BOOL_TO_UINT(eWeightPackage2PhasePackageState[2].bFormPresent);



IF GVL.nFormTransportersScrewerVelocitySV <1000 AND NOT brtLongDelayFirstDraging  THEN
	tonFourthFormat2PhaseSensor.PT:=T#700MS;
ELSIF  (GVL.nFormTransportersScrewerVelocitySV >=1000 AND GVL.nFormTransportersScrewerVelocitySV <1300) AND NOT brtLongDelayFirstDraging THEN
	tonFourthFormat2PhaseSensor.PT:=T#500MS;
ELSIF (GVL.nFormTransportersScrewerVelocitySV >=1300)AND NOT brtLongDelayFirstDraging THEN
	tonFourthFormat2PhaseSensor.PT:=T#300MS;
ELSIF  brtLongDelayFirstDraging THEN
	 tonFourthFormat2PhaseSensor.PT:=T#1000MS;
END_IF

tonDragAE1(IN:=tonDelayAfterStart.Q AND NOT bPhaseChanging AND
		eBeforeDispencer34PackageState2Phase[1].bFormPresent AND eBeforeDispencer34PackageState2Phase[2].bFormPresent AND 
		NOT eAfterDispencer34PackageState2Phase[1].bFormPresent AND NOT eAfterDispencer34PackageState2Phase[2].bFormPresent AND 
		NOT eBeforeDispencer12PackageState2Phase[1].bFormPresent AND NOT eBeforeDispencer12PackageState2Phase[2].bFormPresent 
		,PT:=T#10S);
		
IF tonDelayAfterStart.Q AND NOT bPhaseChanging THEN //Czas po którym możemy przejść do cyklu
	
	//Mamy 4 Formatki w rejestrze przed Dozownikami
	//Pierwszy ruch testy
	IF	 
		//eBeforeDispencer34PackageState2Phase[1].bFormPresent AND eBeforeDispencer34PackageState2Phase[2].bFormPresent AND 
		//NOT eAfterDispencer34PackageState2Phase[1].bFormPresent AND NOT eAfterDispencer34PackageState2Phase[2].bFormPresent AND 
		//NOT eBeforeDispencer12PackageState2Phase[1].bFormPresent AND NOT eBeforeDispencer12PackageState2Phase[2].bFormPresent AND 
		tonDragAE1.Q AND
		NOT P02_Dispencers.fbDispencersDragRightStation.bCycleDone AND NOT P02_Dispencers.fbDispencersDragLeftStation.bCycleDone THEN
		
	   	//4 Formatka stoi na czujniku prze czas T
		IF tonFourthFormat2PhaseSensor.Q  AND NOT (P00_PackML.fbPMLAuto.ePMLState = E_PMLState.ePMLState_STOPPING) (*AND tonCheckFormSensorBetweenDispencer.Q*) THEN
			//VIS.bFormsDragingRightRun							:= TRUE;
			bFormsDragingRightRunCheck							:= TRUE;
			//VIS.bFormsDragingLeftRun							:= TRUE;		//nowe po resecie	
		END_IF
	END_IF
	
(*	
	// Autonaprawa jak się coś rozsypie to przeciągnij lewy
	IF	
		((	eBeforeDispencer12PackageState2Phase[1].bFormPresent	AND	eBeforeDispencer12PackageState2Phase[2].bFormPresent)	OR tonSecondForm2PhaseSensorRepair.Q) AND 
			eAfterDispencer34PackageState2Phase[1].bFormPresent		AND	eAfterDispencer34PackageState2Phase[2].bFormPresent AND 
		NOT eAfterDispencer12PackageState2Phase[1].bFormPresent AND NOT eAfterDispencer12PackageState2Phase[2].bFormPresent AND 
		NOT P02_Dispencers.fbDispencersDragRightStation.bCycleDone AND NOT P02_Dispencers.fbDispencersDragLeftStation.bCycleDone THEN
		
	   	//4 Formatka stoi na czujniku prze czas T
		IF tonFourthFormat2PhaseSensor.Q	 AND NOT (P00_PackML.fbPMLAuto.ePMLState = E_PMLState.ePMLState_STOPPING) (*AND tonCheckFormSensorBetweenDispencer.Q*) THEN
			VIS.bFormsDragingLeftRun							:= TRUE;
		END_IF
	END_IF
*)	
								//200 - Blokada od naprawy gdy formatka wpuszczana jest po jeden
	IF NOT (iGateDispCase=200) AND
		eBeforeDispencer34PackageState2Phase[1].bFormPresent AND eBeforeDispencer34PackageState2Phase[2].bFormPresent AND 
		eBeforeDispencer12PackageState2Phase[1].bFormPresent AND eBeforeDispencer12PackageState2Phase[2].bFormPresent AND 
		NOT P02_Dispencers.fbDispencersDragRightStation.bCycleDone AND NOT P02_Dispencers.fbDispencersDragLeftStation.bCycleDone THEN
		
	   	//4 Formatka stoi na czujniku prze czas T
		IF tonFourthFormat2PhaseSensor.Q AND tonSecondForm2PhaseSensor.Q  AND NOT (P00_PackML.fbPMLAuto.ePMLState = E_PMLState.ePMLState_STOPPING) (*AND tonCheckFormSensorBetweenDispencer.Q*) THEN
			GVL.bFormsDragingRightPrepareRun							:= TRUE;
			GVL.bFormsDragingLeftPrepareRun								:= TRUE; //dodane
		END_IF
		
	
		IF 
		   (eDispencer12PackageState2Phase[1].bFormPresent AND  (eDispencer12PackageState2Phase[1].bDosedSecondPhase OR  eDispencer12PackageState2Phase[1].bDoseAbortedSecondPhase OR NOT eDispencer12PackageState2Phase[1].bBottlePresent)) AND
		   (eDispencer12PackageState2Phase[2].bFormPresent AND  (eDispencer12PackageState2Phase[2].bDosedSecondPhase OR  eDispencer12PackageState2Phase[2].bDoseAbortedSecondPhase OR NOT eDispencer12PackageState2Phase[2].bBottlePresent)) AND
		   (eDispencer34PackageState2Phase[1].bFormPresent AND  (eDispencer34PackageState2Phase[1].bDosed OR  eDispencer34PackageState2Phase[1].bDoseAborted OR NOT eDispencer34PackageState2Phase[1].bBottlePresent)) AND
		   (eDispencer34PackageState2Phase[2].bFormPresent AND  (eDispencer34PackageState2Phase[2].bDosed OR  eDispencer34PackageState2Phase[2].bDoseAborted OR NOT eDispencer34PackageState2Phase[2].bBottlePresent))
		THEN
				//itestdpvs:=itestdpvs+1;
		   	//Rejest za dozownikamu pusty i możemy przeciągać
			IF  NOT eAfterDispencer12PackageState2Phase[1].bFormPresent AND NOT eAfterDispencer12PackageState2Phase[2].bFormPresent	AND
				NOT eAfterDispencer34PackageState2Phase[1].bFormPresent AND NOT eAfterDispencer34PackageState2Phase[2].bFormPresent	AND
				NOT	(P05_Weight.eWeightStation2PhaseRunningState = E_WeightLiftStationState.eRepair)
				THEN
					//itestdpvs2:=itestdpvs2+1;
					//Szlaba zamknięty // dodnae zezwolenie od czujników, bo widły się podnosiły same jak tylko była formatka w rejestrze
					IF P01_Gates.QbGateBeforeDispencersActuator AND 
						(iFormatOnWeight2PhaseCounter < 2 OR NOT VIS.bWeight1EnableShow) AND 
						tonFourthFormat2PhaseSensor.Q AND tonSecondForm2PhaseSensor.Q AND NOT tofWeight6FormSensor.q (*AND VIS.bGateBeforeWeight56Run=FALSE dp ??*) 
						AND NOT tofQueAfterPlatinForDisp.q  AND NOT tonqueafterplatin.q AND NOT tonQueBeforePlatins.q
						AND NOT MAIN.IbSecondFormCheckFormSensor AND NOT P01_Gates.IbGateBeforeWeights56Sensor 
					//(VIS.iNumbersOfFormsBetweenWeightAndScrewers <= P00_PackML.iSetNumbersOfFormsBetweenWeightAndScrewers OR VIS.bWeight1EnableShow)
					//(NOT fbIbCapSorterGateWeightSensor.bOUT OR VIS.bWeight1EnableShow) // dp ZL
					 THEN
					 	//itestdpvs3:=itestdpvs3+1;
						//VIS.bFormsDragingRightRun				:= TRUE;
						//VIS.bFormsDragingLeftRun				:= TRUE; 	
						bFormsDragingLeftRunCheck				:= TRUE;
						bFormsDragingRightRunCheck				:= TRUE;					
					END_IF					
			END_IF 
		END_IF  
	END_IF	
	
	//CycleDone, resetuje pozwolenia
	IF P02_Dispencers.fbDispencersDragRightStation.bCycleDone THEN
		VIS.bFormsDragingRightRun								:= FALSE;
		GVL.bFormsDragingRightPrepareRun						:= FALSE;
		bFormsDragingRightRunCheck								:= FALSE;
	END_IF
	
	//CycleDone, resetuje pozwolenia
	IF P02_Dispencers.fbDispencersDragLeftStation.bCycleDone THEN
		VIS.bFormsDragingLeftRun								:= FALSE;
		GVL.bFormsDragingLeftPrepareRun							:= FALSE;
		bFormsDragingLeftRunCheck								:= FALSE;
	END_IF
	
END_IF

//////////////////////////////////////////////////////////////////////////////////////////////////////
//Test pracy po ESTOP lub Error
IF  NOT bPhaseChanging THEN
	IF P02_Dispencers.fbDispencersDragLeftStation.bWasErrorOrEstop THEN
		IF P02_Dispencers.fbDispencersDragLeftStation.eRunningStateBeforeEStop = E_DragStationState.eDraged OR P02_Dispencers.fbDispencersDragLeftStation.eRunningStateBeforeEStop = E_DragStationState.eEndingOfDrag OR
		   P02_Dispencers.fbDispencersDragLeftStation.eRunningStateBeforeEStop = E_DragStationState.eLowering OR P02_Dispencers.fbDispencersDragLeftStation.eRunningStateBeforeEStop = E_DragStationState.eDraging  THEN
		  //VIS.bFormsDragingLeftRun								:= TRUE;
		   	bFormsDragingLeftRunCheck								:= TRUE;
		END_IF
	END_IF
	
	IF P02_Dispencers.fbDispencersDragRightStation.bWasErrorOrEstop AND NOT bPhaseChanging THEN
		IF P02_Dispencers.fbDispencersDragRightStation.eRunningStateBeforeEStop = E_DragStationState.eDraged OR P02_Dispencers.fbDispencersDragRightStation.eRunningStateBeforeEStop = E_DragStationState.eEndingOfDrag OR
		   P02_Dispencers.fbDispencersDragRightStation.eRunningStateBeforeEStop = E_DragStationState.eLowering OR P02_Dispencers.fbDispencersDragRightStation.eRunningStateBeforeEStop = E_DragStationState.eDraging  THEN	   
		   //VIS.bFormsDragingRightRun								:= TRUE;
		   	bFormsDragingRightRunCheck								:= TRUE;		   
		END_IF
	END_IF
END_IF
END_ACTION

ACTION aP02_DragCheck:
(*
Nazwa:			aP02_DragCheck
Opis:			Zabezpieczenie przeciągania 
Wersja:			v0.2
Data:			2025-06-27
Autor:			DP
Urzadzenia:		
Konfiguracja:	
Info: 
- 
*)

(*Zabezpieczenie przed dozowaniem jak nie złapało formatek i nie znikneły z czujnika*)
MAIN.IbFourthFormCheckFormSensor;	// Czujnik drugiej formatki  przed dozownikami
MAIN.IbSecondFormCheckFormSensor;	// Czujnik czwartek formatki  przed dozownikami
bDispencer12AllowDosingAfterDrag;	// Dodać do VIS.bDispencer1Dose i VIS.bDispencer2Dose
bDispencer34AllowDosingAfterDrag;	// Dodać do VIS.bDispencer3Dose i VIS.bDispencer4Dose

//ftbFormsDragingLeftRun	(CLK:=	P02_Dispencers.fbDispencersDragLeftStation.bCycleDone (*VIS.bFormsDragingLeftRun*),	Q=>); w signals
//ftbFormsDragingRightRun	(CLK:=	P02_Dispencers.fbDispencersDragRightStation.bCycleDone (*VIS.bFormsDragingRightRun*),	Q=>); w signals

IF NOT bDosingTwoPhases AND NOT bPhaseChanging THEN // 1 faza
	IF VIS.bFormsDragingRightRun AND NOT MAIN.IbFourthFormCheckFormSensor THEN
		bDispencer34AllowDosingAfterDrag	:=	TRUE;
	END_IF
	
	IF VIS.bFormsDragingLeftRun  AND NOT MAIN.IbSecondFormCheckFormSensor  THEN
		bDispencer12AllowDosingAfterDrag	:=	TRUE;		
	END_IF
ELSE 						// 2 faza
	;
END_IF



IF (*iDispencersCase = 1 OR iDispencersCase = 3*)rtbFormsDragingLeftRun.q THEN
	bDispencer12AllowDosingAfterDrag	:=	FALSE;	
	bDispencer34AllowDosingAfterDrag	:=	FALSE;
END_IF
(*Koniec Zabezpieczenie przed dozowaniem jak nie złapało formatek i nie znikneły z czujnika*)

(*Sprawdzanie czy mozna zrobić ruch przeciągania*)
IF bFormsDragingLeftEnable AND bFormsDragingRightEnable THEN //Maszyna ma dwufaze
	IF bFormsDragingRightRunCheck  AND (aDispencerLifter34AxisRef.NcToPlc.ActPos + 5) > lrDispencersLifterReadyPosition THEN
		VIS.bFormsDragingRightRun	:= TRUE;
		ibFormsDragingRightRun	:=	ibFormsDragingRightRun	+	1;
	END_IF
	
	IF bFormsDragingLeftRunCheck	AND	(aDispencerLifter12AxisRef.NcToPlc.ActPos + 5) > lrDispencersLifterReadyPosition THEN
		VIS.bFormsDragingLeftRun	:= TRUE;
		ibFormsDragingLeftRun		:=	ibFormsDragingLeftRun	+	1;
	END_IF
ELSE //Maszyna ma tylko 1 przeciąganie
	IF bFormsDragingRightRunCheck  AND	(aDispencerLifter34AxisRef.NcToPlc.ActPos + 5) > lrDispencersLifterReadyPosition AND
										(aDispencerLifter12AxisRef.NcToPlc.ActPos + 5) > lrDispencersLifterReadyPosition 							
	THEN
		VIS.bFormsDragingRightRun	:= TRUE;
		ibFormsDragingRightRun		:=	ibFormsDragingRightRun	+	1;
	END_IF
	
	IF bFormsDragingLeftRunCheck	AND	(aDispencerLifter12AxisRef.NcToPlc.ActPos + 5) > lrDispencersLifterReadyPosition AND
										(aDispencerLifter34AxisRef.NcToPlc.ActPos + 5) > lrDispencersLifterReadyPosition
	THEN
		VIS.bFormsDragingLeftRun	:= TRUE;
		ibFormsDragingLeftRun		:=	ibFormsDragingLeftRun	+	1;
	END_IF
END_IF
END_ACTION

ACTION aP05_Weight:
//Spowolniony transporter
IF bFormTransportersDispencerSlowSpeed THEN
	iWeight56ActuatorUpAddDelay:= 150;
ELSE
	iWeight56ActuatorUpAddDelay:= 0;
END_IF
IF (NOT P00_PackML.bROPPDelayAfterStartFullRegister AND bROPPCappingEnable) OR nFormTransportersScrewerVelocitySV < 400 THEN
	iWeight14ActuatorUpAddDelay:= 275; //bylo 250 a przedtem 150
ELSE
	iWeight14ActuatorUpAddDelay:= 0;
END_IF


tonBreakpoint(IN:=VIS.bWeight1DoWeighting AND eWeightPackageState[1].nCardNumber = 35,PT:=T#5S);
IF tonBreakpoint.Q THEN
	bBreakpoint :=TRUE;
	
END_IF

// Auto Tarowanie po przeważaniu
IF P05_Weight.fbWeightStation.bTareWeights THEN
	VIS.bWeight1Tare := TRUE;
	VIS.bWeight2Tare := TRUE;
	VIS.bWeight3Tare := TRUE;
	VIS.bWeight4Tare := TRUE;
	VIS.bWeight5Tare := NOT bDosingTwoPhases;
	VIS.bWeight6Tare := NOT bDosingTwoPhases;	
ELSE
	VIS.bWeight1Tare := FALSE;
	VIS.bWeight2Tare := FALSE;
	VIS.bWeight3Tare := FALSE;
	VIS.bWeight4Tare := FALSE;	
	VIS.bWeight5Tare := FALSE;
	VIS.bWeight6Tare := FALSE;	
END_IF


(*********** PODNOSZENIE WAG ***********)
(*****************************************)
tonWeight14CycleDoneAndCase(IN:=			// Czasówka na testy
									(
										P05_Weight.fbWeightStation.eRunningState = E_WeightLiftStationState.eRepair OR
										P05_Weight.fbWeightStation.eRunningState = E_WeightLiftStationState.eDisabled OR
										P05_Weight.fbWeightStation.bCycleDone OR 
										P05_Weight.fbWeightStation.eRunningState = E_WeightLiftStationState.eWeighingCycleON OR // Czasami waga czeka na możliwość wypiuszczenia
										(
											P05_Weight.fbWeightStation.eRunningState = E_WeightLiftStationState.eStorageOfForms AND	// Czasami nie ma formatek i czeka na formatki
											NOT eAfterDispencersPackageState[4].bFormPresent									AND
											NOT eAfterDispencersPackageState[3].bFormPresent									AND
											NOT eAfterDispencersPackageState[2].bFormPresent									AND
											NOT eAfterDispencersPackageState[1].bFormPresent											
										)						
									)
									 AND iWeightCase = 30 

, PT:=T#2S);

tonWeight56CycleDoneAndCase(IN:=			// Czasówka na testy
									(
										P05_Weight.fbWeightStation2Phase.eRunningState = E_WeightLiftStationState.eRepair OR
										P05_Weight.fbWeightStation2Phase.eRunningState = E_WeightLiftStationState.eDisabled OR
										P05_Weight.fbWeightStation2Phase.bCycleDone OR 
										P05_Weight.fbWeightStation2Phase.eRunningState = E_WeightLiftStationState.eWeighingCycleON OR // Czasami waga czeka na możliwość wypiuszczenia
										(
											P05_Weight.fbWeightStation2Phase.eRunningState = E_WeightLiftStationState.eStorageOfForms AND	// Czasami nie ma formatek i czeka na formatki
											NOT eAfterDispencer12PackageState2Phase[2].bFormPresent									AND
											NOT eAfterDispencer12PackageState2Phase[1].bFormPresent											
										)						
									)
									 AND iWeightCase = 30 

, PT:=T#2S);

IF tonLongDelayAfterStart.Q THEN

	CASE iWeightCase OF
		
		0:	
		
			IF (
					NOT  bDosingTwoPhases AND ((NOT VIS.bGateBeforeWeight14Run AND NOT P01_Gates.IbGateBeforeWeights14Sensor) OR 
						(
						NOT VIS.bWeightLiftRun AND  P05_Weight.fbWeightStation.bWeight1Actuator AND P05_Weight.fbWeightStation.bWeight2Actuator AND P05_Weight.fbWeightStation.bWeight3Actuator AND  P05_Weight.fbWeightStation.bWeight4Actuator AND P05_Weight.fbWeightStation.bCanReleaseForms
						))
					AND NOT (P00_PackML.fbPMLAuto.ePMLState = E_PMLState.ePMLState_STOPPING)
				) OR  
				(
			  	 bDosingTwoPhases AND NOT VIS.bGateBeforeWeight56Run AND NOT (P00_PackML.fbPMLAuto.ePMLState = E_PMLState.ePMLState_STOPPING)
				)
			THEN
				iWeightCase 				:= iWeightCase	+	10;
			END_IF
			
		10: 
			IF	(NOT  bDosingTwoPhases AND NOT P05_Weight.fbWeightStation.bCycleDone 		AND NOT VIS.bWeightLiftRun) OR
				(	  bDosingTwoPhases AND NOT P05_Weight.fbWeightStation2Phase.bCycleDone	AND NOT 	bWeightLift2PhaseRun) 
			 THEN
				VIS.bWeightLiftRun			:= NOT  bDosingTwoPhases;
					bWeightLift2PhaseRun	:= bDosingTwoPhases;		
					iWeightCase 			:= iWeightCase	+	5;		
			END_IF	
			
		15:
			//(*nie bylo tej linijki*) IF NOT eWeightPackageState[1].bWeighed AND NOT eWeightPackageState[2].bWeighed AND NOT eWeightPackageState[3].bWeighed AND NOT eWeightPackageState[4].bWeighed AND
			 IF P05_Weight.fbWeightStation.eRunningState = E_WeightLiftStationState.eWeighingCycleStart THEN  
				VIS.bWeight1DoWeighting									:= TRUE;
				VIS.bWeight2DoWeighting									:= TRUE;
				VIS.bWeight3DoWeighting									:= TRUE;
				VIS.bWeight4DoWeighting									:= TRUE;
			END_IF
			IF P05_Weight.fbWeightStation2Phase.eRunningState = E_WeightLiftStationState.eWeighingCycleStart THEN 
				VIS.bWeight5DoWeighting									:= TRUE;
				VIS.bWeight6DoWeighting									:= TRUE;
			END_IF	
			IF (NOT  bDosingTwoPhases AND VIS.bWeight1DoWeighting AND VIS.bWeight2DoWeighting AND VIS.bWeight3DoWeighting AND VIS.bWeight4DoWeighting) OR 
					(bDosingTwoPhases AND VIS.bWeight5DoWeighting AND VIS.bWeight6DoWeighting) THEN
				iWeightCase 			:= iWeightCase	+	5;
			END_IF
			
		20: 
			IF	(NOT	bDosingTwoPhases AND P05_Weight.fbWeightStation.bCycleDone) OR
				(		bDosingTwoPhases AND P05_Weight.fbWeightStation2Phase.bCycleDone) 
			THEN
				VIS.bWeightLiftRun			:= FALSE;
					bWeightLift2PhaseRun	:= FALSE;		
					
				VIS.bWeight1DoWeighting		:= FALSE;(*dodane 03.07.2024*)
				VIS.bWeight2DoWeighting		:= FALSE;
				VIS.bWeight3DoWeighting		:= FALSE;
				VIS.bWeight4DoWeighting		:= FALSE;
				VIS.bWeight5DoWeighting		:= FALSE;
				VIS.bWeight6DoWeighting		:= FALSE;(**)				
		
				iWeightCase 				:= 50;
			END_IF				
			IF 
				P05_Weight.fbWeightStation.eRunningState = E_WeightLiftStationState.eRepair	OR 
				P05_Weight.fbWeightStation2Phase.eRunningState = E_WeightLiftStationState.eRepair 
				
				(*VIS.bWeight1DoWeighting		:= FALSE;
				VIS.bWeight2DoWeighting		:= FALSE;
				VIS.bWeight3DoWeighting		:= FALSE;
				VIS.bWeight4DoWeighting		:= FALSE;
				VIS.bWeight5DoWeighting		:= FALSE;
				VIS.bWeight6DoWeighting		:= FALSE;(*CZY TUTAJ TO DODAĆ*)	*)
									
